(* CoDeSys 2.3.9.41 project: КАРАУЛ 10.07.20.pro *)
(* Libraries: Util.lib 18.5.10 15:14:28, UNM.lib 12.9.19 10:56:53, PID_Regulators.lib 12.9.19 10:56:56, STANDARD.LIB 4.10.05 11:14:46, IECSFC.LIB 13.4.06 15:51:28, SYSLIBTIME.LIB 12.9.19 10:55:25, ANALYZATION.LIB 5.10.99 09:05:06 *)

(* PLC configuration (modules and I/O channels)
SBROS_ALL_ERROR AT %IX0.0 [BitInput] DI_1 {ChannellName = Enter name}
AT %IX0.1 [BitInput] DI_2 {ChannellName = Enter name}
B4_GORELKA_1 AT %IX0.2 [BitInput] DI_3 {ChannellName = Enter name}
B4_GORELKA_2 AT %IX0.3 [BitInput] DI_4 {ChannellName = Enter name}
AT %IB1.0 [ByteInput] 8 discrete inputs {ChannellName = Enter name}
AT %IB1.1 [ByteInput] 4 discrete inputs {ChannellName = Enter name}
ESBE_1_LESS AT %QX2.0 [BitOutput] DO_1 {ChannellName = Enter name}
ESBE_1_MORE AT %QX2.1 [BitOutput] DO_2 {ChannellName = Enter name}
ESBE_2_LESS AT %QX2.2 [BitOutput] DO_3 {ChannellName = Enter name}
ESBE_2_MORE AT %QX2.3 [BitOutput] DO_4 {ChannellName = Enter name}
AT %QB3.0 [ByteOutput] 8 discrete outputs {ChannellName = Enter name}
AT %QB3.1 [ByteOutput] 8 signal outputs {ChannellName = Enter name}
Fast analog inputs [ID125] node 4, in %IB4 out %QB4 {ChannellName = Fast analog inputs; Flt_Comm = 50Hz 2Por}
  AT %IR4.0 [FloatInputP] AI #1 {ChannellName = Fast analog input; AIN_TYPE = 4-20 mA; Peak_Filtr = 200; Flt_Ch = Off; TauRC = 10; MinFV = 0; MaxFV = 20000.0}
  AT %IR4.1 [FloatInputP] AI #2 {ChannellName = Fast analog input; AIN_TYPE = 4-20 mA; Peak_Filtr = 200; Flt_Ch = Off; TauRC = 10; MinFV = 0; MaxFV = 20000.0}
  AT %IR4.2 [FloatInputP] AI #3 {ChannellName = Fast analog input; AIN_TYPE = 4-20 mA; Peak_Filtr = 200; Flt_Ch = Off; TauRC = 10; MinFV = 0; MaxFV = 20000.0}
  AT %IR4.3 [FloatInputP] AI #4 {ChannellName = Fast analog input; AIN_TYPE = 4-20 mA; Peak_Filtr = 200; Flt_Ch = Off; TauRC = 10; MinFV = 0; MaxFV = 20000.0}
  AT %IR4.4 [FloatInputP] AI #5 {ChannellName = Fast analog input; AIN_TYPE = 4-20 mA; Peak_Filtr = 200; Flt_Ch = Off; TauRC = 10; MinFV = 0; MaxFV = 20000.0}
  AT %IR4.5 [FloatInputP] AI #6 {ChannellName = Fast analog input; AIN_TYPE = 4-20 mA; Peak_Filtr = 200; Flt_Ch = Off; TauRC = 10; MinFV = 0; MaxFV = 20000.0}
  AT %IR4.6 [FloatInputP] AI #7 {ChannellName = Fast analog input; AIN_TYPE = 4-20 mA; Peak_Filtr = 200; Flt_Ch = Off; TauRC = 10; MinFV = 0; MaxFV = 20000.0}
  AT %IR4.7 [FloatInputP] AI #8 {ChannellName = Fast analog input; AIN_TYPE = 4-20 mA; Peak_Filtr = 200; Flt_Ch = Off; TauRC = 10; MinFV = 0; MaxFV = 20000.0}
  AT %IW4.8 [WordInput] AI read time (10ms) {ChannellName = Enter name}
Analog outputs [ID126] node 5, in %IB5 out %QB5 {ChannellName = Analog outputs}
  AT %QR5.0 [FloatOutputP] AO #1 {ChannellName = Analog output; AOUT_TYPE = 4-20 mA; SafeValueREAL = 0.0}
  AT %QR5.1 [FloatOutputP] AO #2 {ChannellName = Analog output; AOUT_TYPE = 4-20 mA; SafeValueREAL = 0.0}
  AT %QR5.2 [FloatOutputP] AO #3 {ChannellName = Analog output; AOUT_TYPE = 4-20 mA; SafeValueREAL = 0.0}
  AT %QR5.3 [FloatOutputP] AO #4 {ChannellName = Analog output; AOUT_TYPE = 4-20 mA; SafeValueREAL = 0.0}
Special input [ID103] node 6, in %IB6 out %QB6 {ChannellName = Special input}
  AT %IX6.0 [BitInput] Special input {ChannellName = Enter name}
Special output [ID104] node 7, in %IB7 out %QB7 {ChannellName = Special output}
  AT %QX7.0 [BitOutput] Special output {ChannellName = Enter name}
RS-232 [COM2_USART] node 0, in %IB8.0.0 out %QB8.0.0 {ChannellName = RS-232; CommunicationSpeed = 115200; Parity = NO PARITY CHECK; BitLength = 8 bits; StopLength = One stop bit; InterfaceType = RS232; FrameOriented = RTU; Timeout = 0; Visibility = No}
AT %QB8.1.0 [ByteOutput] {ChannellName = Enter name}
AT %QB8.2.0 [ByteOutput] {ChannellName = Enter name}
AT %QB8.3.0 [ByteOutput] {ChannellName = Enter name}
AT %QB8.4.0 [ByteOutput] {ChannellName = Enter name}
AT %QB8.5.0 [ByteOutput] {ChannellName = Enter name}
AT %QB8.6.0 [ByteOutput] {ChannellName = Enter name}
AT %QB8.7.0 [ByteOutput] {ChannellName = Enter name}
AT %QB8.8.0 [ByteOutput] {ChannellName = Enter name}
AT %QB8.9.0 [ByteOutput] {ChannellName = Enter name}
AT %QB8.10.0 [ByteOutput] {ChannellName = Enter name}
AT %QB8.11.0 [ByteOutput] {ChannellName = Enter name}
AT %QB8.12.0 [ByteOutput] {ChannellName = Enter name}
AT %QB8.13.0 [ByteOutput] {ChannellName = Enter name}
AT %QB8.14.0 [ByteOutput] {ChannellName = Enter name}
AT %QB8.15.0 [ByteOutput] {ChannellName = Enter name}
AT %QB8.16.0 [ByteOutput] {ChannellName = Enter name}
AT %QB8.17.0 [ByteOutput] {ChannellName = Enter name}
AT %QB8.18.0 [ByteOutput] {ChannellName = Enter name}
8 bits [8Bit] node 19, in %IB8.19 out %QB8.19 {ChannellName = 8 bit}
  AT %QB8.19.0 [ByteOutput] {ChannellName = Enter name}
8 bits [8Bit] node 20, in %IB8.20 out %QB8.20 {ChannellName = 8 bit}
  AT %QB8.20.0 [ByteOutput] {ChannellName = Enter name}
AVAR_DAVL_PR_OTOP_MAX AT %QD8.21.0 [FloatOutput] {ChannellName = Enter name}
AVAR_DAVL_PR_OTOP_MIN AT %QD8.22.0 [FloatOutput] {ChannellName = Enter name}
USTAVKA_DAVL_OBR_OTOP_ZIMNIY AT %QD8.23.0 [FloatOutput] {ChannellName = Enter name}
PEREPAD_DAVL_OTOP AT %QD8.24.0 [FloatOutput] {ChannellName = Enter name}
AVAR_VREMA_NASOS_OTOPL AT %QD8.25.0 [FloatOutput] {ChannellName = Enter name}
OSNOVNOY_SETEVOY_NASOS AT %QD8.26.0 [FloatOutput] {ChannellName = Enter name}
GISTEREZIS_PODPITKI_OTOPL AT %QD8.27.0 [FloatOutput] {ChannellName = Enter name}
DAVL_POKOYA_OTOP AT %QD8.28.0 [FloatOutput] {ChannellName = Enter name}
Float [Float] node 29, in %IB8.29 out %QB8.29 {ChannellName = float}
  AT %QD8.29.0 [FloatOutput] {ChannellName = Enter name}
Float [Float] node 30, in %IB8.30 out %QB8.30 {ChannellName = float}
  AT %QD8.30.0 [FloatOutput] {ChannellName = Enter name}
Float [Float] node 31, in %IB8.31 out %QB8.31 {ChannellName = float}
  AT %QD8.31.0 [FloatOutput] {ChannellName = Enter name}
Float [Float] node 32, in %IB8.32 out %QB8.32 {ChannellName = float}
  AT %QD8.32.0 [FloatOutput] {ChannellName = Enter name}
  AVAR_DAVL_PR_GVS_MAX AT %QD8.33.0 [FloatOutput] {ChannellName = Enter name}
  AVAR_DAVL_PR_GVS_MIN AT %QD8.34.0 [FloatOutput] {ChannellName = Enter name}
  USTAVKA_DAVL_OBR_GVS AT %QD8.35.0 [FloatOutput] {ChannellName = Enter name}
  PEREPAD_DAVL_GVS AT %QD8.36.0 [FloatOutput] {ChannellName = Enter name}
  AVAR_VREMA_NASOS_GVS AT %QD8.37.0 [FloatOutput] {ChannellName = Enter name}
  OSNOVNOY_GVS_NASOS AT %QD8.38.0 [FloatOutput] {ChannellName = Enter name}
  GISTEREZIS_PODPITKI_GVS AT %QD8.39.0 [FloatOutput] {ChannellName = Enter name}
  DAVL_POKOYA_GVS AT %QD8.40.0 [FloatOutput] {ChannellName = Enter name}
Float [Float] node 41, in %IB8.41 out %QB8.41 {ChannellName = float}
  AT %QD8.41.0 [FloatOutput] {ChannellName = Enter name}
Float [Float] node 42, in %IB8.42 out %QB8.42 {ChannellName = float}
  AT %QD8.42.0 [FloatOutput] {ChannellName = Enter name}
Float [Float] node 43, in %IB8.43 out %QB8.43 {ChannellName = float}
  AT %QD8.43.0 [FloatOutput] {ChannellName = Enter name}
Float [Float] node 44, in %IB8.44 out %QB8.44 {ChannellName = float}
  AT %QD8.44.0 [FloatOutput] {ChannellName = Enter name}
  Float3Module.MODBUS_ID400Parameter.Chan AT %QD8.45.0 [FloatOutput] ellName1Module.FloatfloatfloatSTRINGFloat-IB-%QB-%MB-%M {ChannellName = Enter name}
  Float3Module.MODBUS_ID400Parameter.Chan AT %QD8.46.0 [FloatOutput] ellName1Module.FloatfloatfloatSTRINGFloat.IB.%QB.%MB.%M {ChannellName = Enter name}
Float [Float] node 47, in %IB8.47 out %QB8.47 {ChannellName = float}
  AT %QD8.47.0 [FloatOutput] {ChannellName = Enter name}
Float [Float] node 48, in %IB8.48 out %QB8.48 {ChannellName = float}
  AT %QD8.48.0 [FloatOutput] {ChannellName = Enter name}
  AVAR_VREMA_NASOS_PODPITKI AT %QD8.49.0 [FloatOutput] {ChannellName = Enter name}
  OSNOVNOY_PODPITOCHNIY_NASOS AT %QD8.50.0 [FloatOutput] {ChannellName = Enter name}
Float [Float] node 51, in %IB8.51 out %QB8.51 {ChannellName = float}
  AT %QD8.51.0 [FloatOutput] {ChannellName = Enter name}
Float [Float] node 52, in %IB8.52 out %QB8.52 {ChannellName = float}
  AT %QD8.52.0 [FloatOutput] {ChannellName = Enter name}
Float [Float] node 53, in %IB8.53 out %QB8.53 {ChannellName = float}
  AT %QD8.53.0 [FloatOutput] {ChannellName = Enter name}
Float [Float] node 54, in %IB8.54 out %QB8.54 {ChannellName = float}
  AT %QD8.54.0 [FloatOutput] {ChannellName = Enter name}
Float [Float] node 55, in %IB8.55 out %QB8.55 {ChannellName = float}
  AT %QD8.55.0 [FloatOutput] {ChannellName = Enter name}
Float [Float] node 56, in %IB8.56 out %QB8.56 {ChannellName = float}
  AT %QD8.56.0 [FloatOutput] {ChannellName = Enter name}
  AVAR_DAVL_PR_VNUTR_MAX AT %QD8.57.0 [FloatOutput] {ChannellName = Enter name}
  AVAR_DAVL_PR_VNUTR_MIN AT %QD8.58.0 [FloatOutput] {ChannellName = Enter name}
  USTAVKA_DAVL_OBR_VNUTR AT %QD8.59.0 [FloatOutput] {ChannellName = Enter name}
  PEREPAD_DAVL_VNUTR AT %QD8.60.0 [FloatOutput] {ChannellName = Enter name}
  AVAR_VREMA_NASOS_VNUTR AT %QD8.61.0 [FloatOutput] {ChannellName = Enter name}
  OSNOVNOY_VNUTR_NASOS AT %QD8.62.0 [FloatOutput] {ChannellName = Enter name}
  GISTEREZIS_PODPITKI_VNUTR AT %QD8.63.0 [FloatOutput] {ChannellName = Enter name}
  DAVL_POKOYA_VNUTR AT %QD8.64.0 [FloatOutput] {ChannellName = Enter name}
Float [Float] node 65, in %IB8.65 out %QB8.65 {ChannellName = float}
  AT %QD8.65.0 [FloatOutput] {ChannellName = Enter name}
Float [Float] node 66, in %IB8.66 out %QB8.66 {ChannellName = float}
  AT %QD8.66.0 [FloatOutput] {ChannellName = Enter name}
Float [Float] node 67, in %IB8.67 out %QB8.67 {ChannellName = float}
  AT %QD8.67.0 [FloatOutput] {ChannellName = Enter name}
Float [Float] node 68, in %IB8.68 out %QB8.68 {ChannellName = float}
  AT %QD8.68.0 [FloatOutput] {ChannellName = Enter name}
Float [Float] node 69, in %IB8.69 out %QB8.69 {ChannellName = float}
  VREMYA_RABOTU_CIRCULYACIONNOGO_NASOSA AT %QD8.69.0 [FloatOutput] {ChannellName = Enter name}
Float [Float] node 70, in %IB8.70 out %QB8.70 {ChannellName = float}
  TEMPERATURA_OFF_CIRCULACIONNOGO_NASOSA AT %QD8.70.0 [FloatOutput] {ChannellName = Enter name}
  OSNOVNAYA_GORELKA AT %QD8.71.0 [FloatOutput] {ChannellName = Enter name}
  PODOGREV_2_GORELKOY AT %QD8.72.0 [FloatOutput] {ChannellName = Enter name}
Float [Float] node 73, in %IB8.73 out %QB8.73 {ChannellName = float}
  TEMPERATURA_VKLUCHENIYA_GORELKA_1 AT %QD8.73.0 [FloatOutput] {ChannellName = Enter name}
Float [Float] node 74, in %IB8.74 out %QB8.74 {ChannellName = float}
  TEMPERATURA_OFF_2_STUPENI_GORELKA_1 AT %QD8.74.0 [FloatOutput] {ChannellName = Enter name}
Float [Float] node 75, in %IB8.75 out %QB8.75 {ChannellName = float}
  TEMPERATURA_OFF_TERMOSTAT_GORELKA_1 AT %QD8.75.0 [FloatOutput] {ChannellName = Enter name}
Float [Float] node 76, in %IB8.76 out %QB8.76 {ChannellName = float}
  GISTEREZIS_1_2_STUPEN_GORELKA_1 AT %QD8.76.0 [FloatOutput] {ChannellName = Enter name}
Float [Float] node 77, in %IB8.77 out %QB8.77 {ChannellName = float}
  VREMYA_SBROS_AVARIA_GORELKA_1 AT %QD8.77.0 [FloatOutput] {ChannellName = Enter name}
Float [Float] node 78, in %IB8.78 out %QB8.78 {ChannellName = float}
  TEMPERATURA_AVARIA_MAX_GORELKA_1 AT %QD8.78.0 [FloatOutput] {ChannellName = Enter name}
Float [Float] node 79, in %IB8.79 out %QB8.79 {ChannellName = float}
  AT %QD8.79.0 [FloatOutput] {ChannellName = Enter name}
Float [Float] node 80, in %IB8.80 out %QB8.80 {ChannellName = float}
  AT %QD8.80.0 [FloatOutput] {ChannellName = Enter name}
  PODOGREV_3_GORELKOY AT %QD8.81.0 [FloatOutput] {ChannellName = Enter name}
Float [Float] node 82, in %IB8.82 out %QB8.82 {ChannellName = float}
  TEMPERATURA_VKLUCHENIYA_GORELKA_2 AT %QD8.82.0 [FloatOutput] {ChannellName = Enter name}
Float [Float] node 83, in %IB8.83 out %QB8.83 {ChannellName = float}
  TEMPERATURA_OFF_2_STUPENI_GORELKA_2 AT %QD8.83.0 [FloatOutput] {ChannellName = Enter name}
Float [Float] node 84, in %IB8.84 out %QB8.84 {ChannellName = float}
  TEMPERATURA_OFF_TERMOSTAT_GORELKA_2 AT %QD8.84.0 [FloatOutput] {ChannellName = Enter name}
Float [Float] node 85, in %IB8.85 out %QB8.85 {ChannellName = float}
  GISTEREZIS_1_2_STUPEN_GORELKA_2 AT %QD8.85.0 [FloatOutput] {ChannellName = Enter name}
Float [Float] node 86, in %IB8.86 out %QB8.86 {ChannellName = float}
  VREMYA_SBROS_AVARIA_GORELKA_2 AT %QD8.86.0 [FloatOutput] {ChannellName = Enter name}
  TEMPERATURA_AVARIA_MAX_GORELKA_2 AT %QD8.87.0 [FloatOutput] {ChannellName = Enter name}
Float [Float] node 88, in %IB8.88 out %QB8.88 {ChannellName = float}
  AT %QD8.88.0 [FloatOutput] {ChannellName = Enter name}
Float [Float] node 89, in %IB8.89 out %QB8.89 {ChannellName = float}
  AT %QD8.89.0 [FloatOutput] {ChannellName = Enter name}
Float [Float] node 90, in %IB8.90 out %QB8.90 {ChannellName = float}
  AT %QD8.90.0 [FloatOutput] {ChannellName = Enter name}
Float [Float] node 91, in %IB8.91 out %QB8.91 {ChannellName = float}
  AT %QD8.91.0 [FloatOutput] {ChannellName = Enter name}
Float [Float] node 92, in %IB8.92 out %QB8.92 {ChannellName = float}
  AT %QD8.92.0 [FloatOutput] {ChannellName = Enter name}
Float [Float] node 93, in %IB8.93 out %QB8.93 {ChannellName = float}
  AT %QD8.93.0 [FloatOutput] {ChannellName = Enter name}
Float [Float] node 94, in %IB8.94 out %QB8.94 {ChannellName = float}
  AT %QD8.94.0 [FloatOutput] {ChannellName = Enter name}
Float [Float] node 95, in %IB8.95 out %QB8.95 {ChannellName = float}
  AT %QD8.95.0 [FloatOutput] {ChannellName = Enter name}
Float [Float] node 96, in %IB8.96 out %QB8.96 {ChannellName = float}
  TEMPERATURA_AVARIA_MAX_GORELKA_3 AT %QD8.96.0 [FloatOutput] {ChannellName = Enter name}
Float [Float] node 97, in %IB8.97 out %QB8.97 {ChannellName = float}
  SECOND_GORELKA AT %QD8.97.0 [FloatOutput] {ChannellName = Enter name}
Float [Float] node 98, in %IB8.98 out %QB8.98 {ChannellName = float}
  RESERV_GORELKA AT %QD8.98.0 [FloatOutput] {ChannellName = Enter name}
  GISTEREZIS_PODOGREV AT %QD8.99.0 [FloatOutput] {ChannellName = Enter name}
Float [Float] node 100, in %IB8.100 out %QB8.100 {ChannellName = float}
  AT %QD8.100.0 [FloatOutput] {ChannellName = Enter name}
Float [Float] node 101, in %IB8.101 out %QB8.101 {ChannellName = float}
  AT %QD8.101.0 [FloatOutput] {ChannellName = Enter name}
Float [Float] node 102, in %IB8.102 out %QB8.102 {ChannellName = float}
  AT %QD8.102.0 [FloatOutput] {ChannellName = Enter name}
Float [Float] node 103, in %IB8.103 out %QB8.103 {ChannellName = float}
  AT %QD8.103.0 [FloatOutput] {ChannellName = Enter name}
Float [Float] node 104, in %IB8.104 out %QB8.104 {ChannellName = float}
  AT %QD8.104.0 [FloatOutput] {ChannellName = Enter name}
Float [Float] node 105, in %IB8.105 out %QB8.105 {ChannellName = float}
  AT %QD8.105.0 [FloatOutput] {ChannellName = Enter name}
Float [Float] node 106, in %IB8.106 out %QB8.106 {ChannellName = float}
  AT %QD8.106.0 [FloatOutput] {ChannellName = Enter name}
Float [Float] node 107, in %IB8.107 out %QB8.107 {ChannellName = float}
  AT %QD8.107.0 [FloatOutput] {ChannellName = Enter name}
Float [Float] node 108, in %IB8.108 out %QB8.108 {ChannellName = float}
  AT %QD8.108.0 [FloatOutput] {ChannellName = Enter name}
Float [Float] node 109, in %IB8.109 out %QB8.109 {ChannellName = float}
  AT %QD8.109.0 [FloatOutput] {ChannellName = Enter name}
Float [Float] node 110, in %IB8.110 out %QB8.110 {ChannellName = float}
  AT %QD8.110.0 [FloatOutput] {ChannellName = Enter name}
Float [Float] node 111, in %IB8.111 out %QB8.111 {ChannellName = float}
  AT %QD8.111.0 [FloatOutput] {ChannellName = Enter name}
  EL_2_DAVL_SBROSA_PR_OTOP AT %QD8.112.0 [FloatOutput] {ChannellName = Enter name}
  GISTEREZIS_SBROS_OTOPLENIYA AT %QD8.113.0 [FloatOutput] {ChannellName = Enter name}
Float [Float] node 114, in %IB8.114 out %QB8.114 {ChannellName = float}
  AT %QD8.114.0 [FloatOutput] {ChannellName = Enter name}
  EL_3_DAVL_SBROSA_GVS AT %QD8.115.0 [FloatOutput] {ChannellName = Enter name}
  GISTEREZIS_SBROS_GVS AT %QD8.116.0 [FloatOutput] {ChannellName = Enter name}
Float [Float] node 117, in %IB8.117 out %QB8.117 {ChannellName = float}
  AT %QD8.117.0 [FloatOutput] {ChannellName = Enter name}
Float [Float] node 118, in %IB8.118 out %QB8.118 {ChannellName = float}
  AT %QD8.118.0 [FloatOutput] {ChannellName = Enter name}
Float [Float] node 119, in %IB8.119 out %QB8.119 {ChannellName = float}
  AT %QD8.119.0 [FloatOutput] {ChannellName = Enter name}
Float [Float] node 120, in %IB8.120 out %QB8.120 {ChannellName = float}
  AT %QD8.120.0 [FloatOutput] {ChannellName = Enter name}
Float [Float] node 121, in %IB8.121 out %QB8.121 {ChannellName = float}
  AT %QD8.121.0 [FloatOutput] {ChannellName = Enter name}
Float [Float] node 122, in %IB8.122 out %QB8.122 {ChannellName = float}
  AT %QD8.122.0 [FloatOutput] {ChannellName = Enter name}
Float [Float] node 123, in %IB8.123 out %QB8.123 {ChannellName = float}
  AT %QD8.123.0 [FloatOutput] {ChannellName = Enter name}
Float [Float] node 124, in %IB8.124 out %QB8.124 {ChannellName = float}
  PROPORCIONALNAYA_SOSTAV_ESBE_1 AT %QD8.124.0 [FloatOutput] {ChannellName = Enter name}
Float [Float] node 125, in %IB8.125 out %QB8.125 {ChannellName = float}
  INTEGRALNAYA_SOSTAV_ESBE_1 AT %QD8.125.0 [FloatOutput] {ChannellName = Enter name}
Float [Float] node 126, in %IB8.126 out %QB8.126 {ChannellName = float}
  DIFFERENCIALNAYA_SOSTAV_ESBE_1 AT %QD8.126.0 [FloatOutput] {ChannellName = Enter name}
Float [Float] node 127, in %IB8.127 out %QB8.127 {ChannellName = float}
  VREMYA_HODA_ZADVIZKI_ESBE_1 AT %QD8.127.0 [FloatOutput] {ChannellName = Enter name}
Float [Float] node 128, in %IB8.128 out %QB8.128 {ChannellName = float}
  MIN_VREMYA_OSTANOVKI_ESBE_1 AT %QD8.128.0 [FloatOutput] {ChannellName = Enter name}
Float [Float] node 129, in %IB8.129 out %QB8.129 {ChannellName = float}
  MIN_VREMYA_HODA_ESBE_1 AT %QD8.129.0 [FloatOutput] {ChannellName = Enter name}
  KORREKTIROVKA_USTAVKI_ESBE_1 AT %QD8.130.0 [FloatOutput] {ChannellName = Enter name}
  PROCENT_OTKLONENIA_OT_USTAVKI_ESBE_1 AT %QD8.131.0 [FloatOutput] {ChannellName = Enter name}
  VREMYA_OZIDANIYA_POSLE_SBROSA_ESBE_1 AT %QD8.132.0 [FloatOutput] {ChannellName = Enter name}
  USTAVKA_POSTOYANNAYA_ESBE_1 AT %QD8.133.0 [FloatOutput] {ChannellName = Enter name}
  PROPORCIONALNAYA_SOSTAV_ESBE_2 AT %QD8.134.0 [FloatOutput] {ChannellName = Enter name}
  INTEGRALNAYA_SOSTAV_ESBE_2 AT %QD8.135.0 [FloatOutput] {ChannellName = Enter name}
  DIFFERENCIALNAYA_SOSTAV_ESBE_2 AT %QD8.136.0 [FloatOutput] {ChannellName = Enter name}
  VREMYA_HODA_ZADVIZKI_ESBE_2 AT %QD8.137.0 [FloatOutput] {ChannellName = Enter name}
  MIN_VREMYA_OSTANOVKI_ESBE_2 AT %QD8.138.0 [FloatOutput] {ChannellName = Enter name}
  MIN_VREMYA_HODA_ESBE_2 AT %QD8.139.0 [FloatOutput] {ChannellName = Enter name}
  KORREKTIROVKA_USTAVKI_ESBE_2 AT %QD8.140.0 [FloatOutput] {ChannellName = Enter name}
  PROCENT_OTKLONENIA_OT_USTAVKI_ESBE_2 AT %QD8.141.0 [FloatOutput] {ChannellName = Enter name}
  VREMYA_OZIDANIYA_POSLE_SBROSA_ESBE_2 AT %QD8.142.0 [FloatOutput] {ChannellName = Enter name}
  USTAVKA_POSTOYANNAYA_ESBE_2 AT %QD8.143.0 [FloatOutput] {ChannellName = Enter name}
  BAK_NIGNAYA_GRANICA AT %QD8.144.0 [FloatOutput] {ChannellName = Enter name}
  BAK_VERHNYAY_GRANICA AT %QD8.145.0 [FloatOutput] {ChannellName = Enter name}
  BAK_MIN_PROCENT_AVARIA AT %QD8.146.0 [FloatOutput] {ChannellName = Enter name}
  BAK_MAX_PROCENT_AVARIA AT %QD8.147.0 [FloatOutput] {ChannellName = Enter name}
  BAK_USTAVKA_NAPOLNENIA AT %QD8.148.0 [FloatOutput] {ChannellName = Enter name}
  BAK_GISTEREZIS_NAPOLNENIA AT %QD8.149.0 [FloatOutput] {ChannellName = Enter name}
Float [Float] node 150, in %IB8.150 out %QB8.150 {ChannellName = float}
  AT %QD8.150.0 [FloatOutput] {ChannellName = Enter name}
Float [Float] node 151, in %IB8.151 out %QB8.151 {ChannellName = float}
  AT %QD8.151.0 [FloatOutput] {ChannellName = Enter name}
  NARABOTKA_MINUT_KASKAD_1_NASOS_1_SETEVOY_SP_307 AT %QD8.152.0 [FloatOutput] {ChannellName = Enter name}
  NARABOTKA_MINUT_KASKAD_1_NASOS_2_SETEVOY_SP_307 AT %QD8.153.0 [FloatOutput] {ChannellName = Enter name}
  NARABOTKA_MINUT_KASKAD_3_NASOS_1_GVS_SP_307 AT %QD8.154.0 [FloatOutput] {ChannellName = Enter name}
  NARABOTKA_MINUT_KASKAD_3_NASOS_2_GVS_SP_307 AT %QD8.155.0 [FloatOutput] {ChannellName = Enter name}
  NARABOTKA_MINUT_KASKAD_4_NASOS_1_PODPITKA_SP_307 AT %QD8.156.0 [FloatOutput] {ChannellName = Enter name}
  NARABOTKA_MINUT_KASKAD_4_NASOS_2_PODPITKA_SP_307 AT %QD8.157.0 [FloatOutput] {ChannellName = Enter name}
  NARABOTKA_MINUT_KASKAD_5_NASOS_1_CIRKUL_SP_307 AT %QD8.158.0 [FloatOutput] {ChannellName = Enter name}
  NARABOTKA_MINUT_KASKAD_5_NASOS_2_CIRKUL_SP_307 AT %QD8.159.0 [FloatOutput] {ChannellName = Enter name}
  NARABOTKA_MINUT_GORELKA_1_SP_307 AT %QD8.160.0 [FloatOutput] {ChannellName = Enter name}
Float [Float] node 161, in %IB8.161 out %QB8.161 {ChannellName = float}
  NARABOTKA_MINUT_GORELKA_2_SP_307 AT %QD8.161.0 [FloatOutput] {ChannellName = Enter name}
Float [Float] node 162, in %IB8.162 out %QB8.162 {ChannellName = float}
  NARABOTKA_MINUT_KASKAD_2_VNUTR_NASOS_1_SP_307 AT %QD8.162.0 [FloatOutput] {ChannellName = Enter name}
Float [Float] node 163, in %IB8.163 out %QB8.163 {ChannellName = float}
  NARABOTKA_MINUT_KASKAD_2_VNUTR_NASOS_2_SP_307 AT %QD8.163.0 [FloatOutput] {ChannellName = Enter name}
Float [Float] node 164, in %IB8.164 out %QB8.164 {ChannellName = float}
  NARABOTKA_MINUT_KASKAD_5_NASOS_3_CIRKUL_SP_307 AT %QD8.164.0 [FloatOutput] {ChannellName = Enter name}
Float [Float] node 165, in %IB8.165 out %QB8.165 {ChannellName = float}
  NARABOTKA_MINUT_GORELKA_3_SP_307 AT %QD8.165.0 [FloatOutput] {ChannellName = Enter name}
Float [Float] node 166, in %IB8.166 out %QB8.166 {ChannellName = float}
  KOLICHESTVO_VKLUCHENIY_KASKAD_1_NASOS_1_SETEVOY_SP_307 AT %QD8.166.0 [FloatOutput] {ChannellName = Enter name}
Float [Float] node 167, in %IB8.167 out %QB8.167 {ChannellName = float}
  KOLICHESTVO_VKLUCHENIY_KASKAD_1_NASOS_2_SETEVOY_SP_307 AT %QD8.167.0 [FloatOutput] {ChannellName = Enter name}
Float [Float] node 168, in %IB8.168 out %QB8.168 {ChannellName = float}
  KOLICHESTVO_VKLUCHENIY_KASKAD_3_NASOS_1_GVS_SP_307 AT %QD8.168.0 [FloatOutput] {ChannellName = Enter name}
Float [Float] node 169, in %IB8.169 out %QB8.169 {ChannellName = float}
  KOLICHESTVO_VKLUCHENIY_KASKAD_3_NASOS_2_GVS_SP_307 AT %QD8.169.0 [FloatOutput] {ChannellName = Enter name}
Float [Float] node 170, in %IB8.170 out %QB8.170 {ChannellName = float}
  KOLICHESTVO_VKLUCHENIY_KASKAD_4_NASOS_1_PODPITKA_SP_307 AT %QD8.170.0 [FloatOutput] {ChannellName = Enter name}
Float [Float] node 171, in %IB8.171 out %QB8.171 {ChannellName = float}
  KOLICHESTVO_VKLUCHENIY_KASKAD_4_NASOS_2_PODPITKA_SP_307 AT %QD8.171.0 [FloatOutput] {ChannellName = Enter name}
Float [Float] node 172, in %IB8.172 out %QB8.172 {ChannellName = float}
  KOLICHESTVO_VKLUCHENIY_KASKAD_5_NASOS_1_CIRKUL_SP_307 AT %QD8.172.0 [FloatOutput] {ChannellName = Enter name}
Float [Float] node 173, in %IB8.173 out %QB8.173 {ChannellName = float}
  KOLICHESTVO_VKLUCHENIY_KASKAD_5_NASOS_2_CIRKUL_SP_307 AT %QD8.173.0 [FloatOutput] {ChannellName = Enter name}
Float [Float] node 174, in %IB8.174 out %QB8.174 {ChannellName = float}
  KOLICHESTVO_VKLUCHENIY_GORELKA_1_SP_307 AT %QD8.174.0 [FloatOutput] {ChannellName = Enter name}
Float [Float] node 175, in %IB8.175 out %QB8.175 {ChannellName = float}
  KOLICHESTVO_VKLUCHENIY_GORELKA_2_SP_307 AT %QD8.175.0 [FloatOutput] {ChannellName = Enter name}
Float [Float] node 176, in %IB8.176 out %QB8.176 {ChannellName = float}
  KOLICHESTVO_VKLUCHENIY_KASKAD_2_VNUTR_NASOS_1_SP_307 AT %QD8.176.0 [FloatOutput] {ChannellName = Enter name}
Float [Float] node 177, in %IB8.177 out %QB8.177 {ChannellName = float}
  KOLICHESTVO_VKLUCHENIY_KASKAD_2_VNUTR_NASOS_2_SP_307 AT %QD8.177.0 [FloatOutput] {ChannellName = Enter name}
Float [Float] node 178, in %IB8.178 out %QB8.178 {ChannellName = float}
  KOLICHESTVO_VKLUCHENIY_KASKAD_5_NASOS_3_CIRKUL_SP_307 AT %QD8.178.0 [FloatOutput] {ChannellName = Enter name}
Float [Float] node 179, in %IB8.179 out %QB8.179 {ChannellName = float}
  KOLICHESTVO_VKLUCHENIY_GORELKA_3_SP_307 AT %QD8.179.0 [FloatOutput] {ChannellName = Enter name}
Float [Float] node 180, in %IB8.180 out %QB8.180 {ChannellName = float}
  TEL_KOD_1 AT %QD8.180.0 [FloatOutput] {ChannellName = Enter name}
  TEL_NOMER_1 AT %QD8.181.0 [FloatOutput] {ChannellName = Enter name}
  TEL_KOD_2 AT %QD8.182.0 [FloatOutput] {ChannellName = Enter name}
  TEL_NOMER_2 AT %QD8.183.0 [FloatOutput] {ChannellName = Enter name}
  TEL_KOD_3 AT %QD8.184.0 [FloatOutput] {ChannellName = Enter name}
  TEL_NOMER_3 AT %QD8.185.0 [FloatOutput] {ChannellName = Enter name}
  KOLICESTVO_SOOBSHENIY AT %QD8.186.0 [FloatOutput] {ChannellName = Enter name}
  KOLICHESTVO_NOMEROV AT %QD8.187.0 [FloatOutput] {ChannellName = Enter name}
  TIME_PLANOVAYA_REBBOT_MODEM AT %QD8.188.0 [FloatOutput] {ChannellName = Enter name}
  TIME_WATCH_DOG AT %QD8.189.0 [FloatOutput] {ChannellName = Enter name}
Float [Float] node 190, in %IB8.190 out %QB8.190 {ChannellName = float}
  AT %QD8.190.0 [FloatOutput] {ChannellName = Enter name}
Float [Float] node 191, in %IB8.191 out %QB8.191 {ChannellName = float}
  AT %QD8.191.0 [FloatOutput] {ChannellName = Enter name}
  VREMYA_ZADERGKI_OBRUV_DATCHIKA AT %QD8.192.0 [FloatOutput] {ChannellName = Enter name}
  VREMYA_ZADERGKI_AVARIA_NIZKOE_DAVLENIE AT %QD8.193.0 [FloatOutput] {ChannellName = Enter name}
Float [Float] node 194, in %IB8.194 out %QB8.194 {ChannellName = float}
  AT %QD8.194.0 [FloatOutput] {ChannellName = Enter name}
Float [Float] node 195, in %IB8.195 out %QB8.195 {ChannellName = float}
  AT %QD8.195.0 [FloatOutput] {ChannellName = Enter name}
Float [Float] node 196, in %IB8.196 out %QB8.196 {ChannellName = float}
  AT %QD8.196.0 [FloatOutput] {ChannellName = Enter name}
Float [Float] node 197, in %IB8.197 out %QB8.197 {ChannellName = float}
  AT %QD8.197.0 [FloatOutput] {ChannellName = Enter name}
Float [Float] node 198, in %IB8.198 out %QB8.198 {ChannellName = float}
  TEMPERATURA_1_PR_OTOPLENIYA_AI_SP_307 AT %QD8.198.0 [FloatOutput] {ChannellName = Enter name}
Float [Float] node 199, in %IB8.199 out %QB8.199 {ChannellName = float}
  TEMPERATURA_2_OBR_OTOPLENIYA_AI_SP_307 AT %QD8.199.0 [FloatOutput] {ChannellName = Enter name}
Float [Float] node 200, in %IB8.200 out %QB8.200 {ChannellName = float}
  TEMPERATURA_3_PR_GVS_AI_SP_307 AT %QD8.200.0 [FloatOutput] {ChannellName = Enter name}
Float [Float] node 201, in %IB8.201 out %QB8.201 {ChannellName = float}
  TEMPERATURA_4_OBR_GVS_AI_SP_307 AT %QD8.201.0 [FloatOutput] {ChannellName = Enter name}
Float [Float] node 202, in %IB8.202 out %QB8.202 {ChannellName = float}
  TEMPERATURA_5_KOTEL_1_AI_SP_307 AT %QD8.202.0 [FloatOutput] {ChannellName = Enter name}
Float [Float] node 203, in %IB8.203 out %QB8.203 {ChannellName = float}
  TEMPERATURA_6_KOTEL_2_AI_SP_307 AT %QD8.203.0 [FloatOutput] {ChannellName = Enter name}
Float [Float] node 204, in %IB8.204 out %QB8.204 {ChannellName = float}
  TEMPERATURA_7_KOTEL_3_AI_SP_307 AT %QD8.204.0 [FloatOutput] {ChannellName = Enter name}
Float [Float] node 205, in %IB8.205 out %QB8.205 {ChannellName = float}
  TEMPERATURA_8_ULICA_AI_SP_307 AT %QD8.205.0 [FloatOutput] {ChannellName = Enter name}
Float [Float] node 206, in %IB8.206 out %QB8.206 {ChannellName = float}
  DAVLENIE_1_PR_OTOPLENIYA_AI_SP_307 AT %QD8.206.0 [FloatOutput] {ChannellName = Enter name}
Float [Float] node 207, in %IB8.207 out %QB8.207 {ChannellName = float}
  DAVLENIE_2_OBR_OTOPLENIYA_AI_SP_307 AT %QD8.207.0 [FloatOutput] {ChannellName = Enter name}
Float [Float] node 208, in %IB8.208 out %QB8.208 {ChannellName = float}
  DAVLENIE_3_PR_GVS_AI_SP_307 AT %QD8.208.0 [FloatOutput] {ChannellName = Enter name}
Float [Float] node 209, in %IB8.209 out %QB8.209 {ChannellName = float}
  DAVLENIE_4_OBR_GVS_AI_SP_307 AT %QD8.209.0 [FloatOutput] {ChannellName = Enter name}
Float [Float] node 210, in %IB8.210 out %QB8.210 {ChannellName = float}
  DAVLENIE_5_PR_VNUTR_AI_SP_307 AT %QD8.210.0 [FloatOutput] {ChannellName = Enter name}
Float [Float] node 211, in %IB8.211 out %QB8.211 {ChannellName = float}
  DAVLENIE_6_OBR_VNUTR_AI_SP_307 AT %QD8.211.0 [FloatOutput] {ChannellName = Enter name}
Float [Float] node 212, in %IB8.212 out %QB8.212 {ChannellName = float}
  DAVLENIE_7_NAKOPITELNIY_BAK_AI_SP_307 AT %QD8.212.0 [FloatOutput] {ChannellName = Enter name}
Float [Float] node 213, in %IB8.213 out %QB8.213 {ChannellName = float}
  AT %QD8.213.0 [FloatOutput] {ChannellName = Enter name}
Float [Float] node 214, in %IB8.214 out %QB8.214 {ChannellName = float}
  USTAVKA_ESBE_1_SP_307 AT %QD8.214.0 [FloatOutput] {ChannellName = Enter name}
Float [Float] node 215, in %IB8.215 out %QB8.215 {ChannellName = float}
  USTAVKA_ESBE_2_SP_307 AT %QD8.215.0 [FloatOutput] {ChannellName = Enter name}
Float [Float] node 216, in %IB8.216 out %QB8.216 {ChannellName = float}
  AT %QD8.216.0 [FloatOutput] {ChannellName = Enter name}
Float [Float] node 217, in %IB8.217 out %QB8.217 {ChannellName = float}
  AT %QD8.217.0 [FloatOutput] {ChannellName = Enter name}
Float [Float] node 218, in %IB8.218 out %QB8.218 {ChannellName = float}
  AT %QD8.218.0 [FloatOutput] {ChannellName = Enter name}
Float [Float] node 219, in %IB8.219 out %QB8.219 {ChannellName = float}
  AT %QD8.219.0 [FloatOutput] {ChannellName = Enter name}
2 byte [Register] node 220, in %IB8.220 out %QB8.220 {ChannellName = 2 byte}
  STATUS_NASOS_1_SETEVOY_1_SP_307 AT %QW8.220.0 [WordOutput] {ChannellName = Enter name}
2 byte [Register] node 221, in %IB8.221 out %QB8.221 {ChannellName = 2 byte}
  STATUS_NASOS_2_SETEVOY_1_SP_307 AT %QW8.221.0 [WordOutput] {ChannellName = Enter name}
2 byte [Register] node 222, in %IB8.222 out %QB8.222 {ChannellName = 2 byte}
  STATUS_NASOS_LETNIY_SETEVOY_2_SP_307 AT %QW8.222.0 [WordOutput] {ChannellName = Enter name}
2 byte [Register] node 223, in %IB8.223 out %QB8.223 {ChannellName = 2 byte}
  STATUS_TRUBA_SETEVAYA_SP_307 AT %QW8.223.0 [WordOutput] {ChannellName = Enter name}
2 byte [Register] node 224, in %IB8.224 out %QB8.224 {ChannellName = 2 byte}
  STATUS_NASOS_1_GVS_3_SP_307 AT %QW8.224.0 [WordOutput] {ChannellName = Enter name}
2 byte [Register] node 225, in %IB8.225 out %QB8.225 {ChannellName = 2 byte}
  STATUS_NASOS_2_GVS_3_SP_307 AT %QW8.225.0 [WordOutput] {ChannellName = Enter name}
2 byte [Register] node 226, in %IB8.226 out %QB8.226 {ChannellName = 2 byte}
  STATUS_TRUBA_GVS_SP_307 AT %QW8.226.0 [WordOutput] {ChannellName = Enter name}
2 byte [Register] node 227, in %IB8.227 out %QB8.227 {ChannellName = 2 byte}
  STATUS_NASOS_1_PODPIT_4_SP_307 AT %QW8.227.0 [WordOutput] {ChannellName = Enter name}
2 byte [Register] node 228, in %IB8.228 out %QB8.228 {ChannellName = 2 byte}
  STATUS_NASOS_2_PODPIT_4_SP_307 AT %QW8.228.0 [WordOutput] {ChannellName = Enter name}
2 byte [Register] node 229, in %IB8.229 out %QB8.229 {ChannellName = 2 byte}
  STATUS_TRUBA_PODPITKA_SP_307 AT %QW8.229.0 [WordOutput] {ChannellName = Enter name}
2 byte [Register] node 230, in %IB8.230 out %QB8.230 {ChannellName = 2 byte}
  STATUS_NASOS_1_CIRCULAYCIONNUY_SP_307 AT %QW8.230.0 [WordOutput] {ChannellName = Enter name}
2 byte [Register] node 231, in %IB8.231 out %QB8.231 {ChannellName = 2 byte}
  STATUS_NASOS_2_CIRCULAYCIONNUY_SP_307 AT %QW8.231.0 [WordOutput] {ChannellName = Enter name}
2 byte [Register] node 232, in %IB8.232 out %QB8.232 {ChannellName = 2 byte}
  STATUS_NASOS_3_CIRCULAYCIONNUY_SP_307 AT %QW8.232.0 [WordOutput] {ChannellName = Enter name}
2 byte [Register] node 233, in %IB8.233 out %QB8.233 {ChannellName = 2 byte}
  AT %QW8.233.0 [WordOutput] {ChannellName = Enter name}
2 byte [Register] node 234, in %IB8.234 out %QB8.234 {ChannellName = 2 byte}
  AT %QW8.234.0 [WordOutput] {ChannellName = Enter name}
2 byte [Register] node 235, in %IB8.235 out %QB8.235 {ChannellName = 2 byte}
  AT %QW8.235.0 [WordOutput] {ChannellName = Enter name}
2 byte [Register] node 236, in %IB8.236 out %QB8.236 {ChannellName = 2 byte}
  STATUS_GORELKA1_SP_307 AT %QW8.236.0 [WordOutput] {ChannellName = Enter name}
2 byte [Register] node 237, in %IB8.237 out %QB8.237 {ChannellName = 2 byte}
  STATUS_GORELKA2_SP_307 AT %QW8.237.0 [WordOutput] {ChannellName = Enter name}
2 byte [Register] node 238, in %IB8.238 out %QB8.238 {ChannellName = 2 byte}
  STATUS_GORELKA3_SP_307 AT %QW8.238.0 [WordOutput] {ChannellName = Enter name}
2 byte [Register] node 239, in %IB8.239 out %QB8.239 {ChannellName = 2 byte}
  STATUS_GORENIE_1_B_M_SP_307 AT %QW8.239.0 [WordOutput] {ChannellName = Enter name}
2 byte [Register] node 240, in %IB8.240 out %QB8.240 {ChannellName = 2 byte}
  STATUS_GORENIE_2_B_M_SP_307 AT %QW8.240.0 [WordOutput] {ChannellName = Enter name}
2 byte [Register] node 241, in %IB8.241 out %QB8.241 {ChannellName = 2 byte}
  STATUS_GORENIE_3_B_M_SP_307 AT %QW8.241.0 [WordOutput] {ChannellName = Enter name}
2 byte [Register] node 242, in %IB8.242 out %QB8.242 {ChannellName = 2 byte}
  AT %QW8.242.0 [WordOutput] {ChannellName = Enter name}
2 byte [Register] node 243, in %IB8.243 out %QB8.243 {ChannellName = 2 byte}
  AT %QW8.243.0 [WordOutput] {ChannellName = Enter name}
2 byte [Register] node 244, in %IB8.244 out %QB8.244 {ChannellName = 2 byte}
  AT %QW8.244.0 [WordOutput] {ChannellName = Enter name}
2 byte [Register] node 245, in %IB8.245 out %QB8.245 {ChannellName = 2 byte}
  STATUS_EL_KL_1_PODPITKA_SP_307 AT %QW8.245.0 [WordOutput] {ChannellName = Enter name}
2 byte [Register] node 246, in %IB8.246 out %QB8.246 {ChannellName = 2 byte}
  STATUS_EL_KL_2_SBROS_OTOPLENIAYA_SP_307 AT %QW8.246.0 [WordOutput] {ChannellName = Enter name}
2 byte [Register] node 247, in %IB8.247 out %QB8.247 {ChannellName = 2 byte}
  STATUS_EL_KL_3_SBROS_GVS_SP_307 AT %QW8.247.0 [WordOutput] {ChannellName = Enter name}
  STATUS_EL_KL_4_NAK_BAK_SP_307 AT %QW8.248.0 [WordOutput] {ChannellName = Enter name}
2 byte [Register] node 249, in %IB8.249 out %QB8.249 {ChannellName = 2 byte}
  AT %QW8.249.0 [WordOutput] {ChannellName = Enter name}
2 byte [Register] node 250, in %IB8.250 out %QB8.250 {ChannellName = 2 byte}
  AT %QW8.250.0 [WordOutput] {ChannellName = Enter name}
2 byte [Register] node 251, in %IB8.251 out %QB8.251 {ChannellName = 2 byte}
  AT %QW8.251.0 [WordOutput] {ChannellName = Enter name}
2 byte [Register] node 252, in %IB8.252 out %QB8.252 {ChannellName = 2 byte}
  AT %QW8.252.0 [WordOutput] {ChannellName = Enter name}
2 byte [Register] node 253, in %IB8.253 out %QB8.253 {ChannellName = 2 byte}
  STATUS_BAK_PROCENT_ZAPOLNENIA AT %QW8.253.0 [WordOutput] {ChannellName = Enter name}
2 byte [Register] node 254, in %IB8.254 out %QB8.254 {ChannellName = 2 byte}
  STATUS_ESBE_1_SP_307 AT %QW8.254.0 [WordOutput] {ChannellName = Enter name}
2 byte [Register] node 255, in %IB8.255 out %QB8.255 {ChannellName = 2 byte}
  STATUS_ESBE_2_SP_307 AT %QW8.255.0 [WordOutput] {ChannellName = Enter name}
2 byte [Register] node 256, in %IB8.256 out %QB8.256 {ChannellName = 2 byte}
  STATUS_NASOS_1_VNUTR_2_SP_307 AT %QW8.256.0 [WordOutput] {ChannellName = Enter name}
2 byte [Register] node 257, in %IB8.257 out %QB8.257 {ChannellName = 2 byte}
  STATUS_NASOS_2_VNUTR_2_SP_307 AT %QW8.257.0 [WordOutput] {ChannellName = Enter name}
  STATUS_TRUBA_VNUTR_SP_307 AT %QW8.258.0 [WordOutput] {ChannellName = Enter name}
2 byte [Register] node 259, in %IB8.259 out %QB8.259 {ChannellName = 2 byte}
  AT %QW8.259.0 [WordOutput] {ChannellName = Enter name}
AT %QD9.0 [DWordOutput] Last address {ChannellName = Enter name}
ERROR_CONNECT AT %QW9.1 [WordOutput] Last error {ChannellName = Enter name}
Debug RS-232 [DEBUG_USART] node 0, in %IB9.0 out %QB9.0 {ChannellName = Debug RS-232; CommunicationSpeed = 115200; Parity = NO PARITY CHECK; BitLength = 8 bits; StopLength = One stop bit; InterfaceType = RS232; FrameOriented = ASCII; Timeout = 0; Visibility = No}
Universal Modbus device [ID2000] node 1, in %IB9.1 out %QB9.1 {ChannellName = Universal Modbus device; ModuleIP = 10:0:6:11; ServiceTimeout = 150; TCPport = 502; NetMode = TCP; ModuleSlaveAddress = 1; RequestType = Both; PeriodOfService = 50; Visibility = No; RepeatCounter = 0; ByteSequence = Native}
  AT %QB9.1.0 [ComChannel] Command (0xff - Start) {ChannellName = Enter name}
TEMPERATURA_1_PR_OTOPLENIYA_AI AT %QD9.1.0.0 [FloatOutput] {ChannellName = Enter name}
TEMPERATURA_2_OBR_OTOPLENIYA_AI AT %QD9.1.1.0 [FloatOutput] {ChannellName = Enter name}
TEMPERATURA_3_PR_GVS_AI AT %QD9.1.2.0 [FloatOutput] {ChannellName = Enter name}
TEMPERATURA_4_OBR_GVS_AI AT %QD9.1.3.0 [FloatOutput] {ChannellName = Enter name}
TEMPERATURA_5_KOTEL_1_AI AT %QD9.1.4.0 [FloatOutput] {ChannellName = Enter name}
TEMPERATURA_6_KOTEL_2_AI AT %QD9.1.5.0 [FloatOutput] {ChannellName = Enter name}
TEMPERATURA_7_KOTEL_3_AI AT %QD9.1.6.0 [FloatOutput] {ChannellName = Enter name}
TEMPERATURA_8_ULICA_AI AT %QD9.1.7.0 [FloatOutput] {ChannellName = Enter name}
Universal Modbus device [ID2000] node 2, in %IB9.2 out %QB9.2 {ChannellName = Universal Modbus device; ModuleIP = 10:0:6:12; ServiceTimeout = 150; TCPport = 502; NetMode = TCP; ModuleSlaveAddress = 1; RequestType = Both; PeriodOfService = 50; Visibility = No; RepeatCounter = 0; ByteSequence = Native}
  AT %QB9.2.0 [ComChannel] Command (0xff - Start) {ChannellName = Enter name}
DAVLENIE_1_PR_OTOPLENIYA_AI AT %QD9.2.0.0 [FloatOutput] {ChannellName = Enter name}
DAVLENIE_2_OBR_OTOPLENIYA_AI AT %QD9.2.1.0 [FloatOutput] {ChannellName = Enter name}
DAVLENIE_3_PR_GVS_AI AT %QD9.2.2.0 [FloatOutput] {ChannellName = Enter name}
DAVLENIE_4_OBR_GVS_AI AT %QD9.2.3.0 [FloatOutput] {ChannellName = Enter name}
DAVLENIE_5_PR_VNUTR_AI AT %QD9.2.4.0 [FloatOutput] {ChannellName = Enter name}
DAVLENIE_6_OBR_VNUTR_AI AT %QD9.2.5.0 [FloatOutput] {ChannellName = Enter name}
DAVLENIE_7_NAKOPITELNIY_BAK_AI AT %QD9.2.6.0 [FloatOutput] {ChannellName = Enter name}
AT %QD9.2.7.0 [FloatOutput] {ChannellName = Enter name}
Universal Modbus device [ID2000] node 3, in %IB9.3 out %QB9.3 {ChannellName = Universal Modbus device; ModuleIP = 10:0:6:14; ServiceTimeout = 150; TCPport = 502; NetMode = TCP; ModuleSlaveAddress = 1; RequestType = By poll time; PeriodOfService = 50; Visibility = No; RepeatCounter = 0; ByteSequence = Native}
  AT %QB9.3.0 [ComChannel] Command (0xff - Start) {ChannellName = Enter name}
xDO AT %QW9.3.0.0 [WordOutput] {ChannellName = Enter name}
RS-485-1 [COM1_USART] node 0, in %IB10.0 out %QB10.0 {ChannellName = RS-485-1; CommunicationSpeed = 9600; Parity = NO PARITY CHECK; BitLength = 8 bits; StopLength = One stop bit; InterfaceType = RS485; FrameOriented = ASCII; Timeout = 0; Visibility = No}
*)

(* POU PLC_PRG, ST *)
PROGRAM PLC_PRG
VAR
	I:INT;
	Tpr: REAL; (*-------------------------------------------------------------------------------------ДЛЯ ТЕМПЕРАТУРНОГО РЕЖИМА*)
	T_USTAVKA_T1: REAL;(*--------------------------------------------------------------------УСТАВКА ДЛЯ ПРЯМОЙ ОТОПЛЕНИЯ*)
	T_USTAVKA_T3: REAL;(*------------------------------------------------------------------------------УСТАВКА ДЛЯ ПРЯМОЙ ГВС*)
	PID_OTOPLENIE:PID_REGULATOR;(*---------------------------ПИД РЕГУЛИРОВАНИЕ СМЕСИТЕЛЬНОГО КРАНА ОТОПЛЕНИЕ*)
	PID_GVS:PID_REGULATOR;(*---------------------------------------------ПИД РЕГУЛИРОВАНИЕ СМЕСИТЕЛЬНОГО КРАНА ГВС*)
(*-----------------------------------------------------------------------------------------------------------------------------------------*)
	xDO0,(*---------------------------------------------------------------------------------------------------------НАСОС СЕТЕВОЙ 1*)
	xDO1,(*---------------------------------------------------------------------------------------------------------НАСОС СЕТЕВОЙ 2*)
	xDO2,(*----------------------------------------------------------------------------------------НАСОС ВНУТРЕННЕГО КОНТУРА 1*)
	xDO3,(*----------------------------------------------------------------------------------------НАСОС ВНУТРЕННЕГО КОНТУРА 2*)
	xDO4,(*---------------------------------------------------------------------------------------------------------------НАСОС ГВС 1*)
	xDO5,(*---------------------------------------------------------------------------------------------------------------НАСОС ГВС 2*)
	xDO6,(*--------------------------------------------------------------------------------------------------НАСОС ПОДПИТОЧНЫЙ 1*)
	xDO7,(*--------------------------------------------------------------------------------------------------НАСОС ПОДПИТОЧНЫЙ 2*)
	xDO8,(*----------------------------------------------------------------------------------------------НАСОС ЦИРКУЛЯЦИОННЫЙ 1*)
	xDO9, (*---------------------------------------------------------------------------------------------НАСОС ЦИРКУЛЯЦИОННЫЙ 2*)
	xDO10,(*--------------------------------------------------------------------------------------------НАСОС ЦИРКУЛЯЦИОННЫЙ 3*)
	xDO11,(*-------------------------------------------------------------------------------------------------ГОРЕЛКА 1: ТЕРМОСТАТ*)
	xDO12,(*-------------------------------------------------------------------------------------------------ГОРЕЛКА 2: ТЕРМОСТАТ*)
	xDO13,(*-------------------------------------------------------------------------------------------------ГОРЕЛКА 3: ТЕРМОСТАТ*)
	xDO14,(*------------------------------------------------------------*)
	xDO15:(*------------------------------------------------------------*)
																	   	    BOOL; (*---ЗНАЧЕНИЯ ДИСКРЕТНЫХ МОДУЛЕЙ МУ210-402*)
(*-----------------------------------------------------------------------------------------------------------------------------------------*)

(*-----------------------------------------------------------------------------------ПАРАМЕТРЫ ДЛЯ ВЫЧИСЛЕНИЯ ОШИБКИ МОДУЛЯ*)
	STEP_MODUL_ERROR:INT;
	TIMER_MODUL_ERROR:TP;
(*-----------------------------------------------------------------------------------------------------------------------------------------*)
	NARABOTKA_CHASOV:TON;(*---------------------------------------------------------ТАЙМЕР ДЛЯ НАРАБОТКИ ЧАСОВ/МИНУТ*)
(*---------------------------------------------------------------------------------------------------------ИНИЦИАЛИЗАЦИЯ НАСОСОВ*)



	STEP_ZIMNIY:INT;(*------------------------------------------------------------------------------------------------------------------------------------------УДАЛИТЬ*)
	STEP_LETNIY:INT;(*------------------------------------------------------------------------------------------------------------------------------------------УДАЛИТЬ*)

	KASKAD_NASOSOV_1_SETEVOY:KASKAD_2_NASOSA_2_DATCHIKA_DAVLENIA;
	PUSK_KASKAD_NASOSOV_1_SETEVOY:BOOL;
	WORK_KASKAD_1_SETEVOY:BOOL;(*-----------------------------------------------------------РАБОТА КАСКАДА 1 СЕТЕВОГО*)
	STEP_AVARIA_NIZKOE_DAVLENIE_SETEVOY:INT;
	TIMER_AVARIA_NIZKOE_DAVLENIE_SETEVOY:TP;

	KASKAD_NASOSOV_2_VNUTR:KASKAD_2_NASOSA_2_DATCHIKA_DAVLENIA;
	PUSK_KASKAD_NASOSOV_2_VNUTR:BOOL;
	WORK_KASKAD_2_VNUTR:BOOL;(*-----------------------------------------------------------РАБОТА КАСКАДА 2 ВНУТРЕННЕГО*)
	STEP_AVARIA_NIZKOE_DAVLENIE_VNUTR:INT;
	TIMER_AVARIA_NIZKOE_DAVLENIE_VNUTR:TP;

	KASKAD_NASOSOV_3_GVS:KASKAD_2_NASOSA_2_DATCHIKA_DAVLENIA;
	PUSK_KASKAD_NASOSOV_3_GVS:BOOL;
	WORK_KASKAD_3_GVS:BOOL;(*---------------------------------------------------------------------------РАБОТА КАСКАДА ГВС*)
	STEP_AVARIA_NIZKOE_DAVLENIE_GVS:INT;
	TIMER_AVARIA_NIZKOE_DAVLENIE_GVS:TP;

	KASKAD_NASOSOV_4_PODPITKA:KASKAD_PODPITKA_PO_DATCHIKU_OBRATKI;
	PUSK_KASKAD_NASOSOV_4_PODPITKA:BOOL;
	WORK_KASKAD_4_PODPITKA:BOOL;(*------------------------------------------------------------РАБОТА КАСКАДА ПОДПИТКА*)
	USTAVKA_DAVLENIA_PODPITKA:REAL;(*----------------------------УСТАВКА ОБРАТКИ ДЛЯ ПОДПИТКИ В ЗАВИСИМОСТИ ОТ
																			--------------------------ЗИМНЕГО ИЛИ ЛЕТНЕГО РЕЖИМА*)
(*----------------------------------------------------------------------------------------------------------ИНИЦИАЛИЗАЦИЯ ГОРЕЛОК*)
	GORELKA_1:GORELKA_ROSSEN;
	PUSK_GORELKA_1:BOOL;
	WORK_GORELKA_1:BOOL;(*-----------------------------------------------------------------------------------РАБОТА ГОРЕЛКИ 1*)
	STEP_STATUS_PREDUPREGDENIE_ON_GORELKA_1:INT;
	TIMER_STATUS_PREDUPREGDENIE_ON_GORELKA_1:TP;

	GORELKA_2:GORELKA_ROSSEN;
	PUSK_GORELKA_2:BOOL;
	WORK_GORELKA_2:BOOL;(*-----------------------------------------------------------------------------------РАБОТА ГОРЕЛКИ 2*)
	STEP_STATUS_PREDUPREGDENIE_ON_GORELKA_2:INT;
	TIMER_STATUS_PREDUPREGDENIE_ON_GORELKA_2:TP;

	GORELKA_3:GORELKA_ROSSEN;
	PUSK_GORELKA_3:BOOL;
	WORK_GORELKA_3:BOOL;(*-----------------------------------------------------------------------------------РАБОТА ГОРЕЛКИ 2*)
	STEP_STATUS_PREDUPREGDENIE_ON_GORELKA_3:INT;
	TIMER_STATUS_PREDUPREGDENIE_ON_GORELKA_3:TP;


	AVARIA_OSNOVNAYA_GORELKA:BOOL;
	AVARIA_SECOND_GORELKA:BOOL;
	AVARIA_RESERV_GORELKA:BOOL;

	STEP_PODOGREV_SECOND_GORELKA:INT;
	STEP_PODOGREV_RESERV_GORELKA:INT;
	STEP_AVARIA_PODOGREV_RESERV_GORELKA:INT;

(*----------------------------------------------------------------------------------------ИНИЦИАЛИЗАЦИЯ НАКОПИТЕЛЬНОГО БАКА*)
	BAK:NAKOPITELNYU_BAK;
(*-----------------------------------------------------------------------------------------------------------------------------------------*)

	R_TRIG1: R_TRIG;
	R_TRIG2: R_TRIG;
	R_TRIG3: R_TRIG;
	R_TRIG4: R_TRIG;
	R_TRIG5: R_TRIG;
	R_TRIG6: R_TRIG;
	R_TRIG7: R_TRIG;
	R_TRIG8: R_TRIG;
	R_TRIG9: R_TRIG;
	R_TRIG10: R_TRIG;
	R_TRIG11: R_TRIG;
	R_TRIG12: R_TRIG;
	R_TRIG13: R_TRIG;
	R_TRIG14: R_TRIG;

	DAVLENIE_1_ERROR: BYTE;
	DAVLENIE_2_ERROR: BYTE;
	DAVLENIE_3_ERROR: BYTE;
	DAVLENIE_4_ERROR: BYTE;
	DAVLENIE_5_ERROR: BYTE;
	DAVLENIE_6_ERROR: BYTE;
	DAVLENIE_7_ERROR: BYTE;

	TEMPERATURA_1_ERROR: BYTE;
	TEMPERATURA_2_ERROR: BYTE;
	TEMPERATURA_3_ERROR: BYTE;
	TEMPERATURA_4_ERROR: BYTE;
	TEMPERATURA_5_ERROR: BYTE;
	TEMPERATURA_6_ERROR: BYTE;
	TEMPERATURA_7_ERROR: BYTE;
	TEMPERATURA_8_ERROR: BYTE;

	DAVLENIE_1_DEC: DECODE_FLOAT;
	DAVLENIE_2_DEC: DECODE_FLOAT;
	DAVLENIE_3_DEC: DECODE_FLOAT;
	DAVLENIE_4_DEC: DECODE_FLOAT;
	DAVLENIE_5_DEC: DECODE_FLOAT;
	DAVLENIE_6_DEC: DECODE_FLOAT;
	DAVLENIE_7_DEC: DECODE_FLOAT;
	DAVLENIE_8_DEC: DECODE_FLOAT;

	TEMPERATURA_1_DEC: DECODE_FLOAT;
	TEMPERATURA_2_DEC: DECODE_FLOAT;
	TEMPERATURA_3_DEC: DECODE_FLOAT;
	TEMPERATURA_4_DEC: DECODE_FLOAT;
	TEMPERATURA_5_DEC: DECODE_FLOAT;
	TEMPERATURA_6_DEC: DECODE_FLOAT;
	TEMPERATURA_7_DEC: DECODE_FLOAT;
	TEMPERATURA_8_DEC: DECODE_FLOAT;

	OBRUV_DAVLENIYA_1: OBRYV_DATCHIKA;
	OBRUV_DAVLENIYA_2: OBRYV_DATCHIKA;
	OBRUV_DAVLENIYA_3: OBRYV_DATCHIKA;
	OBRUV_DAVLENIYA_4: OBRYV_DATCHIKA;
	OBRUV_DAVLENIYA_5: OBRYV_DATCHIKA;
	OBRUV_DAVLENIYA_6: OBRYV_DATCHIKA;
	OBRUV_DAVLENIYA_7: OBRYV_DATCHIKA;

	OBRUV_TEMPERATURU_1: OBRYV_DATCHIKA;
	OBRUV_TEMPERATURU_2: OBRYV_DATCHIKA;
	OBRUV_TEMPERATURU_3: OBRYV_DATCHIKA;
	OBRUV_TEMPERATURU_4: OBRYV_DATCHIKA;
	OBRUV_TEMPERATURU_5: OBRYV_DATCHIKA;
	OBRUV_TEMPERATURU_6: OBRYV_DATCHIKA;
	OBRUV_TEMPERATURU_7: OBRYV_DATCHIKA;
	OBRUV_TEMPERATURU_8: OBRYV_DATCHIKA;
(*-----------------------------------------------------------------------------------------------------------------------ОБРЫВ МОДУЛЯ*)
	KOLICHESTVO_OBRUV_MODUL:INT;
(*--------------------------------------------------------------------------------------------------ВСПОМОГАТЕЛЬНЫЙ ПЕРЕМЕННЫЕ*)
	DELTA_TEMPERATURA_USTAVKA:REAL;(*------------РАЗНИЦА МЕЖДУ УСТАВКОЙ И ТЕМПЕРАТУРОЙ ВЫХОДА ОТОПЛЕНИЯ*)
(*--------------------------------------------------------------------------------------------------------------------STEP ОБЪЯВЛЕНИЯ*)
	STEP_MAIN:INT;(*-------------------------------------------------------------------------------------ГЛАВНЫЙ ШАГ АЛГОРИТМА*)
	STEP_DAVL_POKOYA:INT;(*----------------------------------------ДЛЯ ПОДПИТКИ ПЕРЕД ВКЛЮЧЕНИЕМ СЕТЕВЫХ НАСОСОВ*)
	STEP_KASKAD_GVS:INT;(*--------------------------------------------------------------------------------------ДЛЯ ЗАПУСКА ГВС*)
	STEP_KASKAD_GORELKI:INT;(*--------------------------------------------------------------------------ДЛЯ КАСКАДА ГОРЕЛОК*)
	STEP_PODOGREV_2_GORELKOY:INT;(*---------------------------------------------------ДЛЯ ПОДОГРЕВА ВТОРОЙ ГОРЕЛКОЙ*)
	STEP3:INT;(*-------------------------------------------------------------------------ДЛЯ ПЕРЕКЛЮЧЕНИЯ ОСНОВНОЙ ГОРЕЛКИ*)
	STEP4:INT;(*-------------------------------------------------------------------------ДЛЯ ПЕРЕКЛЮЧЕНИЯ ОСНОВНОЙ ГОРЕЛКИ*)
	STEP_CIRCULAYCIONNUY_NASOS_1:INT;(*-----------------------------------ДЛЯ ОТКЛЮЧЕНИЯ ЦИРКУЛЯЦИОННОГО НАСОСА*)
	STEP_CIRCULAYCIONNUY_NASOS_2:INT;(*-----------------------------------ДЛЯ ОТКЛЮЧЕНИЯ ЦИРКУЛЯЦИОННОГО НАСОСА*)
	STEP_CIRCULAYCIONNUY_NASOS_3:INT;(*-----------------------------------ДЛЯ ОТКЛЮЧЕНИЯ ЦИРКУЛЯЦИОННОГО НАСОСА*)
	TIMER_CIRCUL_NASOS_1:TP;
	TIMER_CIRCUL_NASOS_2:TP;
	TIMER_CIRCUL_NASOS_3:TP;
	STEP_PODPITKA_OTOPLENIYA:INT;
	STEP_SBROS_OTOPLENIYA:INT;
	STEP_SBROS_GVS:INT;
	STEP_NAK_BAK:INT;(*-----------------------------------------------------------------------------ДЛЯ НАКОПИТЕЛЬНОГО БАКА*)
END_VAR
VAR RETAIN
(*--------------------------------------------------------------------------------------------------------------------------------АВАРИИ*)
(*'ЭТИ АВАРИИ НУЖНО ОБЪЯВИТЬ ВНУТРИ ПРОГРАММЫ *)
	AVARIA_OBRUV_DATCHIKA_TEMPERATURA_1_PR_OTOP:BOOL;(*-------АВАРИЯ ОБРЫВ ДАТЧИКА Т1 ПРЯМАЯ ОТОПЛЕНИЯ*)
	AVARIA_OBRUV_DATCHIKA_TEMPERATURA_2_OBR_OTOP:BOOL;(*---АВАРИЯ ОБРЫВ ДАТЧИКА Т2 ОБРАТКА ОТОПЛЕНИЯ*)
	AVARIA_OBRUV_DATCHIKA_TEMPERATURA_3_PR_GVS:BOOL;(*------------------АВАРИЯ ОБРЫВ ДАТЧИКА Т3 ПРЯМАЯ ГВС*)
	AVARIA_OBRUV_DATCHIKA_TEMPERATURA_4_OBR_GVS:BOOL;(*---------------АВАРИЯ ОБРЫВ ДАТЧИКА Т4 ОБРАТКА ГВС*)
	AVARIA_OBRUV_DATCHIKA_TEMPERATURA_5_KOTEL_1:BOOL;(*----------------------АВАРИЯ ОБРЫВ ДАТЧИКА Т5 КОТЕЛ 1*)
	AVARIA_OBRUV_DATCHIKA_TEMPERATURA_6_KOTEL_2:BOOL;(*----------------------АВАРИЯ ОБРЫВ ДАТЧИКА Т6 КОТЕЛ 2*)
	AVARIA_OBRUV_DATCHIKA_TEMPERATURA_7_KOTEL_3:BOOL;(*----------------------АВАРИЯ ОБРЫВ ДАТЧИКА Т7 КОТЕЛ 3*)
	AVARIA_OBRUV_DATCHIKA_TEMPERATURA_8_ULICA:BOOL;(*--------------------------АВАРИЯ ОБРЫВ ДАТЧИКА Т7 УЛИЦА*)

	AVARIA_OBRUV_DATCHIKA_DAVLENIE_1_PR_OTOP:BOOL;(*-----------АВАРИЯ ОБРЫВ ДАТЧИКА Р1 ПРЯМАЯ ОТОПЛЕНИЯ*)
	AVARIA_OBRUV_DATCHIKA_DAVLENIE_2_OBR_OTOP:BOOL;(*--------АВАРИЯ ОБРЫВ ДАТЧИКА Р2 ОБРАТКА ОТОПЛЕНИЯ*)
	AVARIA_OBRUV_DATCHIKA_DAVLENIE_3_PR_GVS:BOOL;(*-----------------------АВАРИЯ ОБРЫВ ДАТЧИКА Р3 ПРЯМАЯ ГВС*)
	AVARIA_OBRUV_DATCHIKA_DAVLENIE_4_OBR_GVS:BOOL;(*--------------------АВАРИЯ ОБРЫВ ДАТЧИКА Р4 ОБРАТКА ГВС*)
	AVARIA_OBRUV_DATCHIKA_DAVLENIE_5_PR_VNUTR:BOOL;(*-------------------АВАРИЯ ОБРЫВ ДАТЧИКА Р3 ПРЯМАЯ ВНУТ*)
	AVARIA_OBRUV_DATCHIKA_DAVLENIE_6_OBR_VNUTR:BOOL;(*--------------АВАРИЯ ОБРЫВ ДАТЧИКА Р4 ОБРАТКА ОБРАТ*)
	AVARIA_OBRUV_DATCHIKA_DAVLENIE_7_NAK_BAK:BOOL;(*--------------------------АВАРИЯ ОБРЫВ ДАТЧИКА Р5 НАК.БАК*)

	AVARIA_SETEVOY_NASOS_1:BOOL;(*--------------------------------------------------------------АВАРИЯ СЕТЕВОЙ НАСОС 1*)
	AVARIA_SETEVOY_NASOS_2:BOOL;(*--------------------------------------------------------------АВАРИЯ СЕТЕВОЙ НАСОС 2*)

	AVARIA_VNUTR_NASOS_1:BOOL;(*---------------------------------------------------------------------АВАРИЯ ВНУТР НАСОС 1*)
	AVARIA_VNUTR_NASOS_2:BOOL;(*---------------------------------------------------------------------АВАРИЯ ВНУТР НАСОС 2*)

	AVARIA_GVS_NASOS_1:BOOL;(*---------------------------------------------------------------------------АВАРИЯ НАСОС ГВС 1*)
	AVARIA_GVS_NASOS_2:BOOL;(*---------------------------------------------------------------------------АВАРИЯ НАСОС ГВС 2*)

	AVARIA_PODPITOCHNYU_NASOS_1:BOOL;(*------------------------------------------------АВАРИЯ ПОДПИТОЧНЫЙ НАСОС 1*)
	AVARIA_PODPITOCHNYU_NASOS_2:BOOL;(*------------------------------------------------АВАРИЯ ПОДПИТОЧНЫЙ НАСОС 2*)

	AVARIA_GORELKA_1:BOOL;(*---------------------------------------------------------------------------------АВАРИЯ ГОРЕЛКА 1*)
	AVARIA_GORELKA_2:BOOL;(*---------------------------------------------------------------------------------АВАРИЯ ГОРЕЛКА 2*)
	AVARIA_GORELKA_3:BOOL;(*---------------------------------------------------------------------------------АВАРИЯ ГОРЕЛКА 2*)


END_VAR
VAR (* helpers for the ST form of the networks *)
	_t5 : TIME;
END_VAR
IF BIT_VKLUCHENIYA_SP_307=TRUE THEN (*-----------------------------------------------------------------------БИТ ВКЛЮЧЕНИЯ*)
(*---------------------------------------------------------------------------------------------------------------------------------МОДЕМ*)

MODEM;

(*----------------------------------------------------------------------------------------------------ДИСКРЕТНЫЙ ВЫВОД НА МОДУЛЬ*)
DO_DISKRETNUY_OUT;
(*---------------------------------------------------------------------------------------------------------------------ОБРЫВ ДАТЧИКОВ*)
DECOD_ERROR;
IF PUSK_SP_307 THEN
	AVARIA_DATCHIK;(*---------------------ЧТО БЫ НЕ ЛЕТЕЛИ АВАРИИ ОБРЫВА ДАТЧИКОВ ПОКА КОТЕЛЬНАЯ НЕ ЗАПУЩЕНА*)
END_IF
(*-------------------------------------------------------------------------------------------------------------------НАРАБОТКА МИНУТ*)
NARABOTKA_MINUT;
(*------------------------------------------------------------------------------------------------------------------------ОТВАЛ МОДУЛЯ*)

MODUL_ERROR;

(*-------------------------------------------------------------------------------------------------------------НАРАБОТКА ВКЛЮЧЕНИЙ*)
NARABOTKA_VKLUCHENIY;
(*--------------------------------------------------------------------------------------------------------ПОГОДОЗАВИСИМЫЙ ГРАФИК*)
TEMPERATURNYU_REGIM;
(*----------------------------------------------------------------------------------------------------АЛГОРИТМ РАБОТЫ КОТЕЛЬНОЙ*)
ALGORITHM;

(*---------------------------------------------------------------------------------------------------------ЦИРКУЛЯЦИОННЫЙ НАСОСЫ*)
CIRCULAYCIONNYE_NASOSU;
(*-------------------------------------------------------------------------------------------------------КАСКАД НАСОСОВ 1 СЕТЕВОЙ*)
KASKAD_NASOSOV_1_SETEVOY(
	OSNOVNOY:=REAL_TO_INT(OSNOVNOY_SETEVOY_NASOS),(*---------------------------------------------ОСНОВНОЙ НАСОС*)
	TIME_AVARIA:=REAL_TO_TIME(AVAR_VREMA_NASOS_OTOPL*1000),(*-----------------------------------ВРЕМЯ НА АВАРИЮ*)
	P_1:=DAVLENIE_1_PR_OTOPLENIYA_AI_SP_307,(*------------------------------------------------ДАВЛЕНИЕ ПОСЛЕ КАСКАДА*)
	P_2:=DAVLENIE_2_OBR_OTOPLENIYA_AI_SP_307, (*--------------------------------------------ДАВЛЕНИЕ ПЕРЕД КАСКАДОМ*)
	PEREPAD_DAVLENIA:=PEREPAD_DAVL_OTOP, (*-----------------------------------------------------------ПЕРЕПАД ДАВЛЕНИЯ*)
	SBROS_ERROR:=SBROS_AVARIA_SETEVOY_KASKAD_1_SP_307, (*---------------------СБРОС ОШИБКИ КАСКАДА НАСОСОВ*)
	PUSK_NASOS:=PUSK_KASKAD_NASOSOV_1_SETEVOY, (*------------------------------------------ПУСК КАСКАДА НАСОСОВ*)
	ERROR_NASOS1:=AVARIA_SETEVOY_NASOS_1, (*----------------ОШИБКА НАСОСА 1. ХРАНИТСЯ В RETAIN КОНТРОЛЛЕРА*)
	ERROR_NASOS2:=AVARIA_SETEVOY_NASOS_2, (*----------------ОШИБКА НАСОСА 2. ХРАНИТСЯ В RETAIN КОНТРОЛЛЕРА*)
	RELE_NASOS1=>xDO0, (*---------------------------------------------------------------------------РЕЛЕ ВКЛЮЧЕНИЯ НАСОСА 1*)
	RELE_NASOS2=>xDO1, (*---------------------------------------------------------------------------РЕЛЕ ВКЛЮЧЕНИЯ НАСОСА 2*)
	WORK=>WORK_KASKAD_1_SETEVOY,(*--------------------------------------------------СТАТУС РАБОТА КАСКАДА НАСОСОВ*)
);
(*--------------------------------------------------------------------------------------------------------КАСКАД НАСОСОВ 2 ЛЕТНИЙ*)
KASKAD_NASOSOV_2_VNUTR(
	OSNOVNOY:=REAL_TO_INT(OSNOVNOY_VNUTR_NASOS),(*---------------------------------------------ОСНОВНОЙ НАСОС*)
	TIME_AVARIA:=REAL_TO_TIME(AVAR_VREMA_NASOS_VNUTR*1000),(*-----------------------------------ВРЕМЯ НА АВАРИЮ*)
	P_1:=DAVLENIE_5_PR_VNUTR_AI_SP_307,(*------------------------------------------------ДАВЛЕНИЕ ПОСЛЕ КАСКАДА*)
	P_2:=DAVLENIE_6_OBR_VNUTR_AI_SP_307, (*--------------------------------------------ДАВЛЕНИЕ ПЕРЕД КАСКАДОМ*)
	PEREPAD_DAVLENIA:=PEREPAD_DAVL_VNUTR, (*-----------------------------------------------------------ПЕРЕПАД ДАВЛЕНИЯ*)
	SBROS_ERROR:=SBROS_AVARIA_VNUTR_KASKAD_2_SP_307, (*---------------------СБРОС ОШИБКИ КАСКАДА НАСОСОВ*)
	PUSK_NASOS:=PUSK_KASKAD_NASOSOV_2_VNUTR, (*------------------------------------------ПУСК КАСКАДА НАСОСОВ*)
	ERROR_NASOS1:=AVARIA_VNUTR_NASOS_1, (*----------------ОШИБКА НАСОСА 1. ХРАНИТСЯ В RETAIN КОНТРОЛЛЕРА*)
	ERROR_NASOS2:=AVARIA_VNUTR_NASOS_2, (*----------------ОШИБКА НАСОСА 2. ХРАНИТСЯ В RETAIN КОНТРОЛЛЕРА*)
	RELE_NASOS1=>xDO2, (*---------------------------------------------------------------------------РЕЛЕ ВКЛЮЧЕНИЯ НАСОСА 1*)
	RELE_NASOS2=>xDO3, (*---------------------------------------------------------------------------РЕЛЕ ВКЛЮЧЕНИЯ НАСОСА 2*)
	WORK=>WORK_KASKAD_2_VNUTR,(*--------------------------------------------------СТАТУС РАБОТА КАСКАДА НАСОСОВ*)
);
(*-------------------------------------------------------------------------------------------------------------КАСКАД НАСОСОВ 3 ГВС*)
KASKAD_NASOSOV_3_GVS(
	OSNOVNOY:=REAL_TO_INT(OSNOVNOY_GVS_NASOS),(*---------------------------------------------------ОСНОВНОЙ НАСОС*)
	TIME_AVARIA:=REAL_TO_TIME(AVAR_VREMA_NASOS_GVS*1000),(*--------------------------------------ВРЕМЯ НА АВАРИЮ*)
	P_1:=DAVLENIE_3_PR_GVS_AI_SP_307,(*----------------------------------------------------------ДАВЛЕНИЕ ПОСЛЕ КАСКАДА*)
	P_2:=DAVLENIE_4_OBR_GVS_AI_SP_307, (*------------------------------------------------------ДАВЛЕНИЕ ПЕРЕД КАСКАДОМ*)
	PEREPAD_DAVLENIA:=PEREPAD_DAVL_GVS, (*-------------------------------------------------------------ПЕРЕПАД ДАВЛЕНИЯ*)
	SBROS_ERROR:=SBROS_AVARIA_GVS_KASKAD_3_SP_307, (*---------------------------СБРОС ОШИБКИ КАСКАДА НАСОСОВ*)
	PUSK_NASOS:=PUSK_KASKAD_NASOSOV_3_GVS, (*-------------------------------------------------ПУСК КАСКАДА НАСОСОВ*)
	ERROR_NASOS1:=AVARIA_GVS_NASOS_1, (*----------------------ОШИБКА НАСОСА 1. ХРАНИТСЯ В RETAIN КОНТРОЛЛЕРА*)
	ERROR_NASOS2:=AVARIA_GVS_NASOS_2, (*----------------------ОШИБКА НАСОСА 2. ХРАНИТСЯ В RETAIN КОНТРОЛЛЕРА*)
	RELE_NASOS1=>xDO4, (*---------------------------------------------------------------------------РЕЛЕ ВКЛЮЧЕНИЯ НАСОСА 1*)
	RELE_NASOS2=>xDO5, (*---------------------------------------------------------------------------РЕЛЕ ВКЛЮЧЕНИЯ НАСОСА 2*)
	WORK=>WORK_KASKAD_3_GVS(*---------------------------------------------------------СТАТУС РАБОТА КАСКАДА НАСОСОВ*)
);
(*----------------------------------------------------------------------------------------------КАСКАД ПОДПИТОЧНЫЙХ НАСОСОВ 4*)
(*------В ЗАВИСИМОСТИ ОТ ТОГО В КАКОМ РЕЖИМЕ РАБОТАЕТ КОТЕЛЬНАЯ (ЗИМНИЙ ИЛИ ЛЕТНИЙ) БЕРЕТСЯ УСТАВКА ДЛЯ *)
(*-------------------------------------------------------------------------------ПОДПИТКИ ОТ КОТОРОЙ ОТСЧИТЫВАЕТСЯ АВАРИЯ*)

USTAVKA_DAVLENIA_PODPITKA:=USTAVKA_DAVL_OBR_OTOP_ZIMNIY;(*----------------------------------УСТАВКА ПОДПИТКИ*)

(*IF LETNIY_KASKAD_PUSK_SP_307 THEN USTAVKA_DAVLENIA_PODPITKA:=USTAVKA_DAVL_OBR_LETNIY; END_IF ----------------------------------------------------------------УДАЛИТЬ*)

KASKAD_NASOSOV_4_PODPITKA(
	OSNOVNOY:=REAL_TO_INT(OSNOVNOY_PODPITOCHNIY_NASOS),(*-------------------------------------ОСНОВНОЙ НАСОС*)
	TIME_AVARIA:=REAL_TO_TIME(AVAR_VREMA_NASOS_PODPITKI*1000),(*-------------------------------ВРЕМЯ НА АВАРИЮ*)
	P:=DAVLENIE_2_OBR_OTOPLENIYA_AI_SP_307,(*-----------------------ДАВЛЕНИЕ ОБРАТКИ ПОДПИТЫВАЕМОГО КОНТУРА*)
	USTAVKA_P:=USTAVKA_DAVLENIA_PODPITKA, (*-----------------------------------------------------------УСТАВКА ОБРАТКИ*)(*<------------------------------------------ ВОТ ЭТОТ ПАРАМЕТР НУЖНО НА ЗИМНИЙ И ЛЕТНИЙ РАЗВЕСТИ, ДАВЛЕНИЯ БУДУТ РАЗНЫЕ*)
	SBROS_ERROR:=SBROS_AVARIA_PODPITOCHNY_KASKAD_4_SP_307, (*---------------СБРОС ОШИБКИ КАСКАДА НАСОСОВ*) (*--------------------------------------------ДОБАВИЛ , НАДО ПРОВЕРЯТЬ*)
	PUSK_NASOS:=PUSK_KASKAD_NASOSOV_4_PODPITKA, (*------------------------------------------ПУСК КАСКАДА НАСОСОВ*)
	ERROR_NASOS1:=AVARIA_PODPITOCHNYU_NASOS_1, (*---------ОШИБКА НАСОСА 1. ХРАНИТСЯ В RETAIN КОНТРОЛЛЕРА*)
	ERROR_NASOS2:=AVARIA_PODPITOCHNYU_NASOS_2, (*---------ОШИБКА НАСОСА 2. ХРАНИТСЯ В RETAIN КОНТРОЛЛЕРА*)
	RELE_NASOS1=>xDO6, (*---------------------------------------------------------------------------РЕЛЕ ВКЛЮЧЕНИЯ НАСОСА 1*)
	RELE_NASOS2=>xDO7, (*---------------------------------------------------------------------------РЕЛЕ ВКЛЮЧЕНИЯ НАСОСА 2*)
	WORK=>WORK_KASKAD_4_PODPITKA,(*-------------------------------------------------СТАТУС РАБОТА КАСКАДА НАСОСОВ*)
);
(*------------------------------------------------------------------------------------------------ТРЕХХОДОВОЙ КРАН ОТОПЛЕНИЕ  1*)
IF PUSK_ESBE_SP_307 THEN
PID_OTOPLENIE(
	USTAVKA:=T_USTAVKA_T1,
	KORREKTIROVKA:=KORREKTIROVKA_USTAVKI_ESBE_1,
	SBROS:=SBROS_ESBE_1_SP_307,
	TEMPERATURA_IN:=TEMPERATURA_1_PR_OTOPLENIYA_AI_SP_307,
	ESBE_VREMYA_HODA_ZADVIGKI:=VREMYA_HODA_ZADVIZKI_ESBE_1,
	ESBE_MIN_VREMYA_HODA:=MIN_VREMYA_HODA_ESBE_1,
	ESBE_MIN_VREMYA_OSTANOVKI:=MIN_VREMYA_OSTANOVKI_ESBE_1,
	ESBE_PROPORCIONAL:=PROPORCIONALNAYA_SOSTAV_ESBE_1,
	ESBE_INTEGRAL:=INTEGRALNAYA_SOSTAV_ESBE_1,
	ESBE_DIFFERINCAL:=DIFFERENCIALNAYA_SOSTAV_ESBE_1,
	LESS=>ESBE_1_LESS,
	MORE=>ESBE_1_MORE,
);
END_IF
(*----------------------------------------------------------------------------------------------------------ТРЕХХОДОВОЙ КРАН ГВС  2*)
T_USTAVKA_T3:=USTAVKA_POSTOYANNAYA_ESBE_2+KORREKTIROVKA_USTAVKI_ESBE_2;
IF PUSK_ESBE_SP_307 THEN
PID_GVS(
	USTAVKA:=USTAVKA_POSTOYANNAYA_ESBE_2,
	KORREKTIROVKA:=KORREKTIROVKA_USTAVKI_ESBE_2,
	SBROS:=SBROS_ESBE_2_SP_307,
	TEMPERATURA_IN:=TEMPERATURA_3_PR_GVS_AI_SP_307,
	ESBE_VREMYA_HODA_ZADVIGKI:=VREMYA_HODA_ZADVIZKI_ESBE_2,
	ESBE_MIN_VREMYA_HODA:=MIN_VREMYA_HODA_ESBE_2,
	ESBE_MIN_VREMYA_OSTANOVKI:=MIN_VREMYA_OSTANOVKI_ESBE_2,
	ESBE_PROPORCIONAL:=PROPORCIONALNAYA_SOSTAV_ESBE_2,
	ESBE_INTEGRAL:=INTEGRALNAYA_SOSTAV_ESBE_2,
	ESBE_DIFFERINCAL:=DIFFERENCIALNAYA_SOSTAV_ESBE_2,
	LESS=>ESBE_2_LESS,
	MORE=>ESBE_2_MORE,
);
END_IF
(*-----------------------------------------------------------------------------------------------------------------------------ГОРЕЛКА 1*)
GORELKA_1(
	PUSK:=PUSK_GORELKA_1,
	TEMPERATURA_KOTLA:=TEMPERATURA_5_KOTEL_1_AI_SP_307,
	AVARIA:=S3_GORELKA_1,(*---------------------------------------------------------------------------------ОШИБКА С ГОРЕЛКИ 220 В*)
	AVAR_TEMPERATURA:=TEMPERATURA_AVARIA_MAX_GORELKA_1,
	SBROS_ERROR:=SBROS_AVARIA_GORELKA_1_SP_307,(*---------------------------------------------СБРОС АВАРИИ ГОРЕЛКИ*)
	ERROR_GORELKA:=AVARIA_GORELKA_1,(*------------------------------------------------------------------------------АВАРИЯ ГОРЕЛКА 1*)
	TERM=>xDO11,(*----------------------------------------------------------------------------------КЛЕММЫ ЗАПРОС НА РОЗЖИГ*)
	WORK=>WORK_GORELKA_1,(*-------------------------------------------------------------------------СТАТУС РАБОТА ГОРЕЛКИ*)
);
(*----------------------------------------------------------------------------------------------------------------------------ГОРЕЛКА 2*)
GORELKA_2(
	PUSK:=PUSK_GORELKA_2,
	TEMPERATURA_KOTLA:=TEMPERATURA_6_KOTEL_2_AI_SP_307,
	AVARIA:=S3_GORELKA_2,(*---------------------------------------------------------------------------------ОШИБКА С ГОРЕЛКИ 220 В*)
	AVAR_TEMPERATURA:=TEMPERATURA_AVARIA_MAX_GORELKA_2,
	SBROS_ERROR:=SBROS_AVARIA_GORELKA_2_SP_307,(*---------------------------------------------СБРОС АВАРИИ ГОРЕЛКИ*)
	ERROR_GORELKA:=AVARIA_GORELKA_2,(*------------------------------------------------------------------------------АВАРИЯ ГОРЕЛКА 1*)
	TERM=>xDO12,(*----------------------------------------------------------------------------------КЛЕММЫ ЗАПРОС НА РОЗЖИГ*)
	WORK=>WORK_GORELKA_2,(*-------------------------------------------------------------------------СТАТУС РАБОТА ГОРЕЛКИ*)
);
(*----------------------------------------------------------------------------------------------------------------------------ГОРЕЛКА 3*)
GORELKA_3(
	PUSK:=PUSK_GORELKA_3,
	TEMPERATURA_KOTLA:=TEMPERATURA_7_KOTEL_3_AI_SP_307,
	AVARIA:=S3_GORELKA_3,(*---------------------------------------------------------------------------------ОШИБКА С ГОРЕЛКИ 220 В*)
	AVAR_TEMPERATURA:=TEMPERATURA_AVARIA_MAX_GORELKA_3,
	SBROS_ERROR:=SBROS_AVARIA_GORELKA_3_SP_307,(*---------------------------------------------СБРОС АВАРИИ ГОРЕЛКИ*)
	ERROR_GORELKA:=AVARIA_GORELKA_3,(*------------------------------------------------------------------------------АВАРИЯ ГОРЕЛКА 1*)
	TERM=>xDO13,(*----------------------------------------------------------------------------------КЛЕММЫ ЗАПРОС НА РОЗЖИГ*)
	WORK=>WORK_GORELKA_3,(*-------------------------------------------------------------------------СТАТУС РАБОТА ГОРЕЛКИ*)
);
(*----------------------------------------------------------------------------------------------------------------НАКОПИТЕЛЬНЫЙ БАК*)
BAK(
	P:=DAVLENIE_7_NAKOPITELNIY_BAK_AI_SP_307,(*--------------------------ДАВЛЕНИЕ ДАТЧИКА НАКОПИТЕЛЬНОГО БАКА*)
	D_MIN:=BAK_NIGNAYA_GRANICA,(*-----------------------------------------------------------ДАВЛЕНИЕ МИНИМАЛЬНОЕ В 0%*)
	D_MAX:=BAK_VERHNYAY_GRANICA,(*-----------------------------------------------------ДАВЛЕНИЕ МАКСИМАЛЬНОЕ В 100%*)
	PROCENT_ZAPOLNENIA=>STATUS_BAK_PROCENT_ZAPOLNENIA, (*----------------------------------ПРОЦЕНТ ЗАПОЛНЕНИЯ*)
);
(*-----------------------------------------------------------------------------------------------------------------------------------------*)

(*----СБРОС ОШИБОК ДОЛЖЕН ВЫПОЛНЯТЬСЯ В САМОМ КОНЦЕ ПОСЛЕ ИНИЦИАЛИЗАЦИЙ ВСЕХ ФУНКЦИОНАЛЬНЫХ БЛОКОВ*)
(*-----------------------------------------------------------------------------------------------------------------ОБРАБОТКА АВАРИЙ*)

IF PUSK_SP_307 THEN
	AVARIA_STATUS;
END_IF

(*-----------------------------------------------------------------------------------------------------------------ОБРАБОТКА АВАРИЙ*)

OBRABOTKA_AVARIY;

(*-----------------------------------------------------------------------------------------------------------------------СБРОС ОШИБОК*)

SBROS_ERROR;
(*-----------------------------------------------------------------------------------СТАТУСЫ ЭЛЕМЕНТОВ КОТЕЛЬНОЙ ДЛЯ ПАНЕЛИ*)
OUT_STATUS_SP_307;
END_IF (*--------------------------------------------------------------------------------------------------------------БИТ ВКЛЮЧЕНИЯ*)
END_PROGRAM
ACTION ALGORITHM:
(*----------------------------------------------------------------------------------------------------------------НАКОПИТЕЛЬНЫЙ БАК*)
IF STATUS_BAK_PROCENT_ZAPOLNENIA<BAK_USTAVKA_NAPOLNENIA AND STEP_NAK_BAK=0  THEN
	STEP_NAK_BAK:=1;
END_IF
CASE STEP_NAK_BAK OF
	1:
		EL_KL_4_NAK_BAK:=TRUE; (*-------------------------------------------------------------ВКЛЮЧАЕМ КЛАПАН НАКОПИТЕЛЬНОГО БАКА*)
		IF STATUS_BAK_PROCENT_ZAPOLNENIA>=BAK_USTAVKA_NAPOLNENIA+BAK_GISTEREZIS_NAPOLNENIA THEN
			STEP_NAK_BAK:=2;
		END_IF
	2:
		EL_KL_4_NAK_BAK:=FALSE; (*-----------------------------------------------------------ОТКЛЮЧАЕМ КЛАПАН НАКОПИТЕЛЬНОГО БАКА*)
		STEP_NAK_BAK:=0;
END_CASE





(*------------------------------------------------------------------РАСЧЕТ ОТКЛОНЕНИЯ ТЕМПЕРАТУРЫ ОТОПЛЕНИЯ ОТ УСТАВКИ*)
DELTA_TEMPERATURA_USTAVKA:=T_USTAVKA_T1-TEMPERATURA_1_PR_OTOPLENIYA_AI_SP_307;
(*-----------------------------------------------------------------------------------------------------------------------------------------*)



(*------------------------ЕСЛИ ПУСК КОТЕЛЬНАЯ НАЖАТА  И МОДУЛИ НЕ ОТВАЛИЛИСЬ ТО НАЧИНАЕМ ВЫПОЛНЯТЬ АЛГОРИТМ*)
(*----------------------------------------------------------------------------------------------------------------ЗАПУСК НАСОСОВ ГВС*)
IF PUSK_SP_307=TRUE AND ERROR_MODUL_SP_307=FALSE AND AVARIA_PHASA_SP_307=FALSE AND PUSK_GVS_SP_307
AND AVARIA_VUSOKOE_DAVLENIE_GVS_SP_307=FALSE AND AVARIA_NIZKOE_DAVLENIE_GVS_SP_307=FALSE AND AVARIA_FIRE_SP_307=FALSE AND AVARIA_GAZ_SP_307=FALSE  THEN
	IF AVARIA_GVS_NASOS_1=FALSE OR AVARIA_GVS_NASOS_2=FALSE THEN
		PUSK_KASKAD_NASOSOV_3_GVS:=TRUE;
	ELSE
		PUSK_KASKAD_NASOSOV_3_GVS:=FALSE;
	END_IF
ELSE
	PUSK_KASKAD_NASOSOV_3_GVS:=FALSE;
	xDO.4:=xDO4:=FALSE;(*---------------------------------------------------------------------------------------------НАСОС ГВС 1*)
	xDO.5:=xDO5:=FALSE;(*---------------------------------------------------------------------------------------------НАСОС ГВС 2*)
END_IF


IF PUSK_SP_307=TRUE AND ERROR_MODUL_SP_307=FALSE AND AVARIA_PHASA_SP_307=FALSE AND VNUTR_KASKAD_PUSK_SP_307
(*AND AVARIA_VUSOKOE_DAVLENIE_OTOPLENIYA_SP_307=FALSE AND AVARIA_NIZKOE_DAVLENIE_OTOPLENIYA_SP_307=FALSE AND STEP_MAIN>101*)  THEN
	IF AVARIA_VNUTR_NASOS_1=FALSE OR AVARIA_VNUTR_NASOS_2=FALSE  THEN
		PUSK_KASKAD_NASOSOV_2_VNUTR:=TRUE;
	ELSE
		PUSK_KASKAD_NASOSOV_2_VNUTR:=FALSE;
	END_IF
ELSE
	PUSK_KASKAD_NASOSOV_2_VNUTR:=FALSE;
	xDO.2:=xDO2:=FALSE;(*-------------------------------------------------------------------------------НАСОС ВНУТР.КОНТУРА 1*)
	xDO.3:=xDO3:=FALSE;(*-------------------------------------------------------------------------------НАСОС ВНУТР.КОНТУРА 2*)
END_IF

(*--------------------------------------------------------------------------------------------------------------СБРОС ОТОПЛЕНИЯ*)
	IF DAVLENIE_1_PR_OTOPLENIYA_AI_SP_307>EL_2_DAVL_SBROSA_PR_OTOP
  	 AND STEP_SBROS_OTOPLENIYA=0 THEN
		STEP_SBROS_OTOPLENIYA:=1;
	END_IF
	CASE STEP_SBROS_OTOPLENIYA OF
		1:
			EL_KL_2_SBROS_OTOPL:=TRUE; (*-----------------------------------------------ВКЛЮЧЕНИЕ КЛАПАНА СБРОСА ОТОПЛЕНИ*)
			IF DAVLENIE_1_PR_OTOPLENIYA_AI_SP_307<=EL_2_DAVL_SBROSA_PR_OTOP-GISTEREZIS_SBROS_OTOPLENIYA THEN
				STEP_SBROS_OTOPLENIYA:=2;
			END_IF
		2:
			EL_KL_2_SBROS_OTOPL:=FALSE; (*----------------------------------------------ВЫКЛЮЧЕНИЕ КЛАПАНА СБРОСА ОТОПЛЕНИЯ*)
			STEP_SBROS_OTOPLENIYA:=0;
	END_CASE

(*--------------------------------------------------------------------------------------------------------------СБРОС ГВС*)
	IF DAVLENIE_3_PR_GVS_AI_SP_307>EL_3_DAVL_SBROSA_GVS
  	 AND STEP_SBROS_GVS=0 THEN
		STEP_SBROS_GVS:=1;
	END_IF
	CASE STEP_SBROS_GVS OF
		1:
			EL_KL_3_SBROS_GVS:=TRUE; (*-----------------------------------------------ВКЛЮЧЕНИЕ КЛАПАНА СБРОСА ОТОПЛЕНИ*)
			IF DAVLENIE_3_PR_GVS_AI_SP_307<=EL_3_DAVL_SBROSA_GVS-GISTEREZIS_SBROS_GVS THEN
				STEP_SBROS_GVS:=2;
			END_IF
		2:
			EL_KL_3_SBROS_GVS:=FALSE; (*----------------------------------------------ВЫКЛЮЧЕНИЕ КЛАПАНА СБРОСА ОТОПЛЕНИЯ*)
			STEP_SBROS_GVS:=0;
	END_CASE



(*--------------------------------------------------------------------------------------------------------------ПОДПИТКА ОТОПЛЕНИЯ*)
	IF DAVLENIE_2_OBR_OTOPLENIYA_AI_SP_307<USTAVKA_DAVL_OBR_OTOP_ZIMNIY AND WORK_KASKAD_1_SETEVOY
  	 AND STEP_PODPITKA_OTOPLENIYA=0
	AND (AVARIA_PODPITOCHNYU_NASOS_1=FALSE OR AVARIA_PODPITOCHNYU_NASOS_2=FALSE)THEN
		STEP_PODPITKA_OTOPLENIYA:=1;
	END_IF
	CASE STEP_PODPITKA_OTOPLENIYA OF
		1:
			EL_KL_1_PODPITKA_OTOPL:=TRUE; (*-----------------------------------------------ВКЛЮЧЕНИЕ КЛАПАНА ПОДПИТКИ*)
			PUSK_KASKAD_NASOSOV_4_PODPITKA:=TRUE;
			IF DAVLENIE_2_OBR_OTOPLENIYA_AI_SP_307>=USTAVKA_DAVL_OBR_OTOP_ZIMNIY+GISTEREZIS_PODPITKI_OTOPL THEN
				STEP_PODPITKA_OTOPLENIYA:=2;
			END_IF
			IF  AVARIA_PODPITOCHNYU_NASOS_1  AND AVARIA_PODPITOCHNYU_NASOS_2  THEN
				STEP_PODPITKA_OTOPLENIYA:=2;
			END_IF
			IF WORK_KASKAD_1_SETEVOY=FALSE OR (AVARIA_SETEVOY_NASOS_1
			AND AVARIA_SETEVOY_NASOS_2) THEN
				STEP_PODPITKA_OTOPLENIYA:=2;
			END_IF
		2:
			EL_KL_1_PODPITKA_OTOPL:=FALSE; (*----------------------------------------------ВКЛЮЧЕНИЕ КЛАПАНА ПОДПИТКИ*)
			PUSK_KASKAD_NASOSOV_4_PODPITKA:=FALSE;
			STEP_PODPITKA_OTOPLENIYA:=0;
	END_CASE




(*--------------------------------------------------------------------------------------------------------ЗАПУСК СЕТЕВОГО КОНТУРА*)
IF PUSK_SP_307=TRUE AND ERROR_MODUL_SP_307=FALSE AND AVARIA_PHASA_SP_307=FALSE
AND AVARIA_VUSOKOE_DAVLENIE_OTOPLENIYA_SP_307=FALSE
AND AVARIA_NIZKOE_DAVLENIE_OTOPLENIYA_SP_307=FALSE  THEN
	CASE STEP_MAIN OF
		0: 						(*-------------------------------------------------------------------------------------ВКЛЮЧЕНИЕ ГАЗА*)
			(*xDO11:=TRUE;*)(*--------------------------------------------------------------------------------------------------------------------------КЛАПАНА ГАЗА НЕТ*)
			STEP_MAIN:=100;
		100:	                   (*-------ПЕРВОНАЧАЛЬНАЯ ПОДПИТКА ПРЯМОЙ ОТОПЛЕНИЯ ПЕРЕД ЗАПУСКОМ СЕТЕВЫХ НАСОСОВ*)
			IF (DAVLENIE_1_PR_OTOPLENIYA_AI<DAVL_POKOYA_OTOP) AND FIRST_START_SP_307  THEN
				STEP_MAIN:=101;
				STEP_DAVL_POKOYA:=1;
			ELSE
				STEP_MAIN:=110;
				STEP_KASKAD_GVS:=10;
			END_IF
		101: (*----------------------------------------------------------------------ПОДПИТЫВАЕМ СЕТЕВОЙ КОНТУР ДО УСТАВКИ*)
			CASE STEP_DAVL_POKOYA OF
				1:
					IF DAVLENIE_1_PR_OTOPLENIYA_AI<DAVL_POKOYA_OTOP THEN
						EL_KL_1_PODPITKA_OTOPL:=TRUE;  (*--------------------------------ВКЛЮЧЕНИЕ ЭЛЕКТРОКЛАПАНА 1 ПОДПИТКИ ОТОПЛЕНИЯ*)
					END_IF
					STEP_DAVL_POKOYA:=2;
				2:
					PUSK_KASKAD_NASOSOV_4_PODPITKA:=TRUE;
					IF AVARIA_PODPITOCHNYU_NASOS_1 AND AVARIA_PODPITOCHNYU_NASOS_2 THEN
						STEP_DAVL_POKOYA:=4;
					END_IF
					IF DAVLENIE_1_PR_OTOPLENIYA_AI>DAVL_POKOYA_OTOP THEN
						EL_KL_1_PODPITKA_OTOPL:=FALSE;  (*-----------------------------ВЫКЛЮЧЕНИЕ ЭЛЕКТРОКЛАПАНА 1 ПОДПИТКИ ОТОПЛЕНИЯ*)
					ELSE
						EL_KL_1_PODPITKA_OTOPL:=TRUE;  (*--------------------------------ВКЛЮЧЕНИЕ ЭЛЕКТРОКЛАПАНА 1 ПОДПИТКИ ОТОПЛЕНИЯ*)
					END_IF

					IF DAVLENIE_1_PR_OTOPLENIYA_AI>DAVL_POKOYA_OTOP THEN
						STEP_DAVL_POKOYA:=3;
					END_IF
				3:
					PUSK_KASKAD_NASOSOV_4_PODPITKA:=FALSE;
					EL_KL_1_PODPITKA_OTOPL:=FALSE;  (*---------------------------------ВЫКЛЮЧЕНИЕ ЭЛЕКТРОКЛАПАНА 1 ПОДПИТКИ ОТОПЛЕНИЯ*)
					STEP_MAIN:=110;
					STEP_KASKAD_GVS:=10;
					STEP_DAVL_POKOYA:=0;
				4:
					PUSK_KASKAD_NASOSOV_4_PODPITKA:=FALSE;
					EL_KL_1_PODPITKA_OTOPL:=FALSE;  (*---------------------------------ВЫКЛЮЧЕНИЕ ЭЛЕКТРОКЛАПАНА 1 ПОДПИТКИ ОТОПЛЕНИЯ*)
			END_CASE
		110:(*-------------------------------------------------------------------------------------------ЗАПУСК СЕТЕВОГО КАСКАДА*)

				PUSK_KASKAD_NASOSOV_1_SETEVOY:=TRUE;


			IF WORK_KASKAD_1_SETEVOY  THEN
				KASKAD_GORELOK;(*--------------------------------------------------------------------ЗАПУСК КАСКАДА ГОРЕЛОК*)
			ELSE
				PUSK_GORELKA_1:=FALSE;
				PUSK_GORELKA_2:=FALSE;
				PUSK_GORELKA_3:=FALSE;
			END_IF
	END_CASE






ELSE(*------------------ЕСЛИ ПУСК КОТЕЛЬНАЯ НАЖАТА  И МОДУЛИ НЕ ОТВАЛИЛИСЬ ТО НАЧИНАЕМ ВЫПОЛНЯТЬ АЛГОРИТМ*)



	xDO.0:=xDO0:=FALSE;(*---------------------------------------------------------------------------------------НАСОС СЕТЕВОЙ 1*)
	xDO.1:=xDO1:=FALSE;(*---------------------------------------------------------------------------------------НАСОС СЕТЕВОЙ 2*)
(*
	xDO.2:=xDO2:=FALSE;(*----------------------------------------------------------------------------------НАСОС ВНУТРЕННИЙ 1*)
	xDO.3:=xDO3:=FALSE;(*----------------------------------------------------------------------------------НАСОС ВНУТРЕННИЙ 2*)
	xDO.4:=xDO4:=FALSE;(*-----------------------------------------------------------------------------------------НАСОС ГВС 1*)
	xDO.5:=xDO5:=FALSE;(*-----------------------------------------------------------------------------------------НАСОС ГВС 2*)
*)
	xDO.6:=xDO6:=FALSE;(*--------------------------------------------------------------------------------НАСОС ПОДПИТОЧНЫЙ 1*)
	xDO.7:=xDO7:=FALSE;(*--------------------------------------------------------------------------------НАСОС ПОДПИТОЧНЫЙ 2*)
	(*xDO.8:=xDO8:=FALSE;*)(*-----------------------------------------------------------------------НАСОС ЦИРКУЛЯЦИОННЫЙ 1*)
	(*xDO.9:=xDO9:=FALSE;*)(*-----------------------------------------------------------------------НАСОС ЦИРКУЛЯЦИОННЫЙ 2*)
	(*xDO.10:=xDO10:=FALSE;*)(*--------------------------------------------------------------------НАСОС ЦИРКУЛЯЦИОННЫЙ 3*)
	xDO.11:=xDO11:=FALSE;(*----------------------------------------------------------------------------------КОТЕЛ ТЕРМОСТАТ 1*)
	xDO.12:=xDO12:=FALSE;(*----------------------------------------------------------------------------------КОТЕЛ ТЕРМОСТАТ 2*)
	xDO.13:=xDO13:=FALSE;(*----------------------------------------------------------------------------------КОТЕЛ ТЕРМОСТАТ 3*)
	xDO.14:=xDO14:=FALSE;(*----------------------------------------------------------------------------------------------------------*)
	xDO.15:=xDO15:=FALSE;(*----------------------------------------------------------------------------------------------------------*)

	PUSK_GORELKA_1:=FALSE;
	PUSK_GORELKA_2:=FALSE;
	PUSK_GORELKA_3:=FALSE;
	PUSK_KASKAD_NASOSOV_1_SETEVOY:=FALSE;
	(*PUSK_KASKAD_NASOSOV_2_VNUTR:=FALSE;*)
	(*PUSK_KASKAD_NASOSOV_3_GVS:=FALSE;*)
	PUSK_KASKAD_NASOSOV_4_PODPITKA:=FALSE;

	STEP_MAIN:=0;
	STEP_DAVL_POKOYA:=0;
	STEP3:=0;
	STEP4:=0;
	(*
	STEP_SBROS_GVS:=0;
	STEP_SBROS_OTOPLENIYA:=0;
	*)
	STEP_PODOGREV_SECOND_GORELKA:=0;
	STEP_PODOGREV_RESERV_GORELKA:=0;
	STEP_AVARIA_PODOGREV_RESERV_GORELKA:=0;
END_IF(*----------------ЕСЛИ ПУСК КОТЕЛЬНАЯ НАЖАТА  И МОДУЛИ НЕ ОТВАЛИЛИСЬ ТО НАЧИНАЕМ ВЫПОЛНЯТЬ АЛГОРИТМ*)
END_ACTION
ACTION AVARIA_DATCHIK:
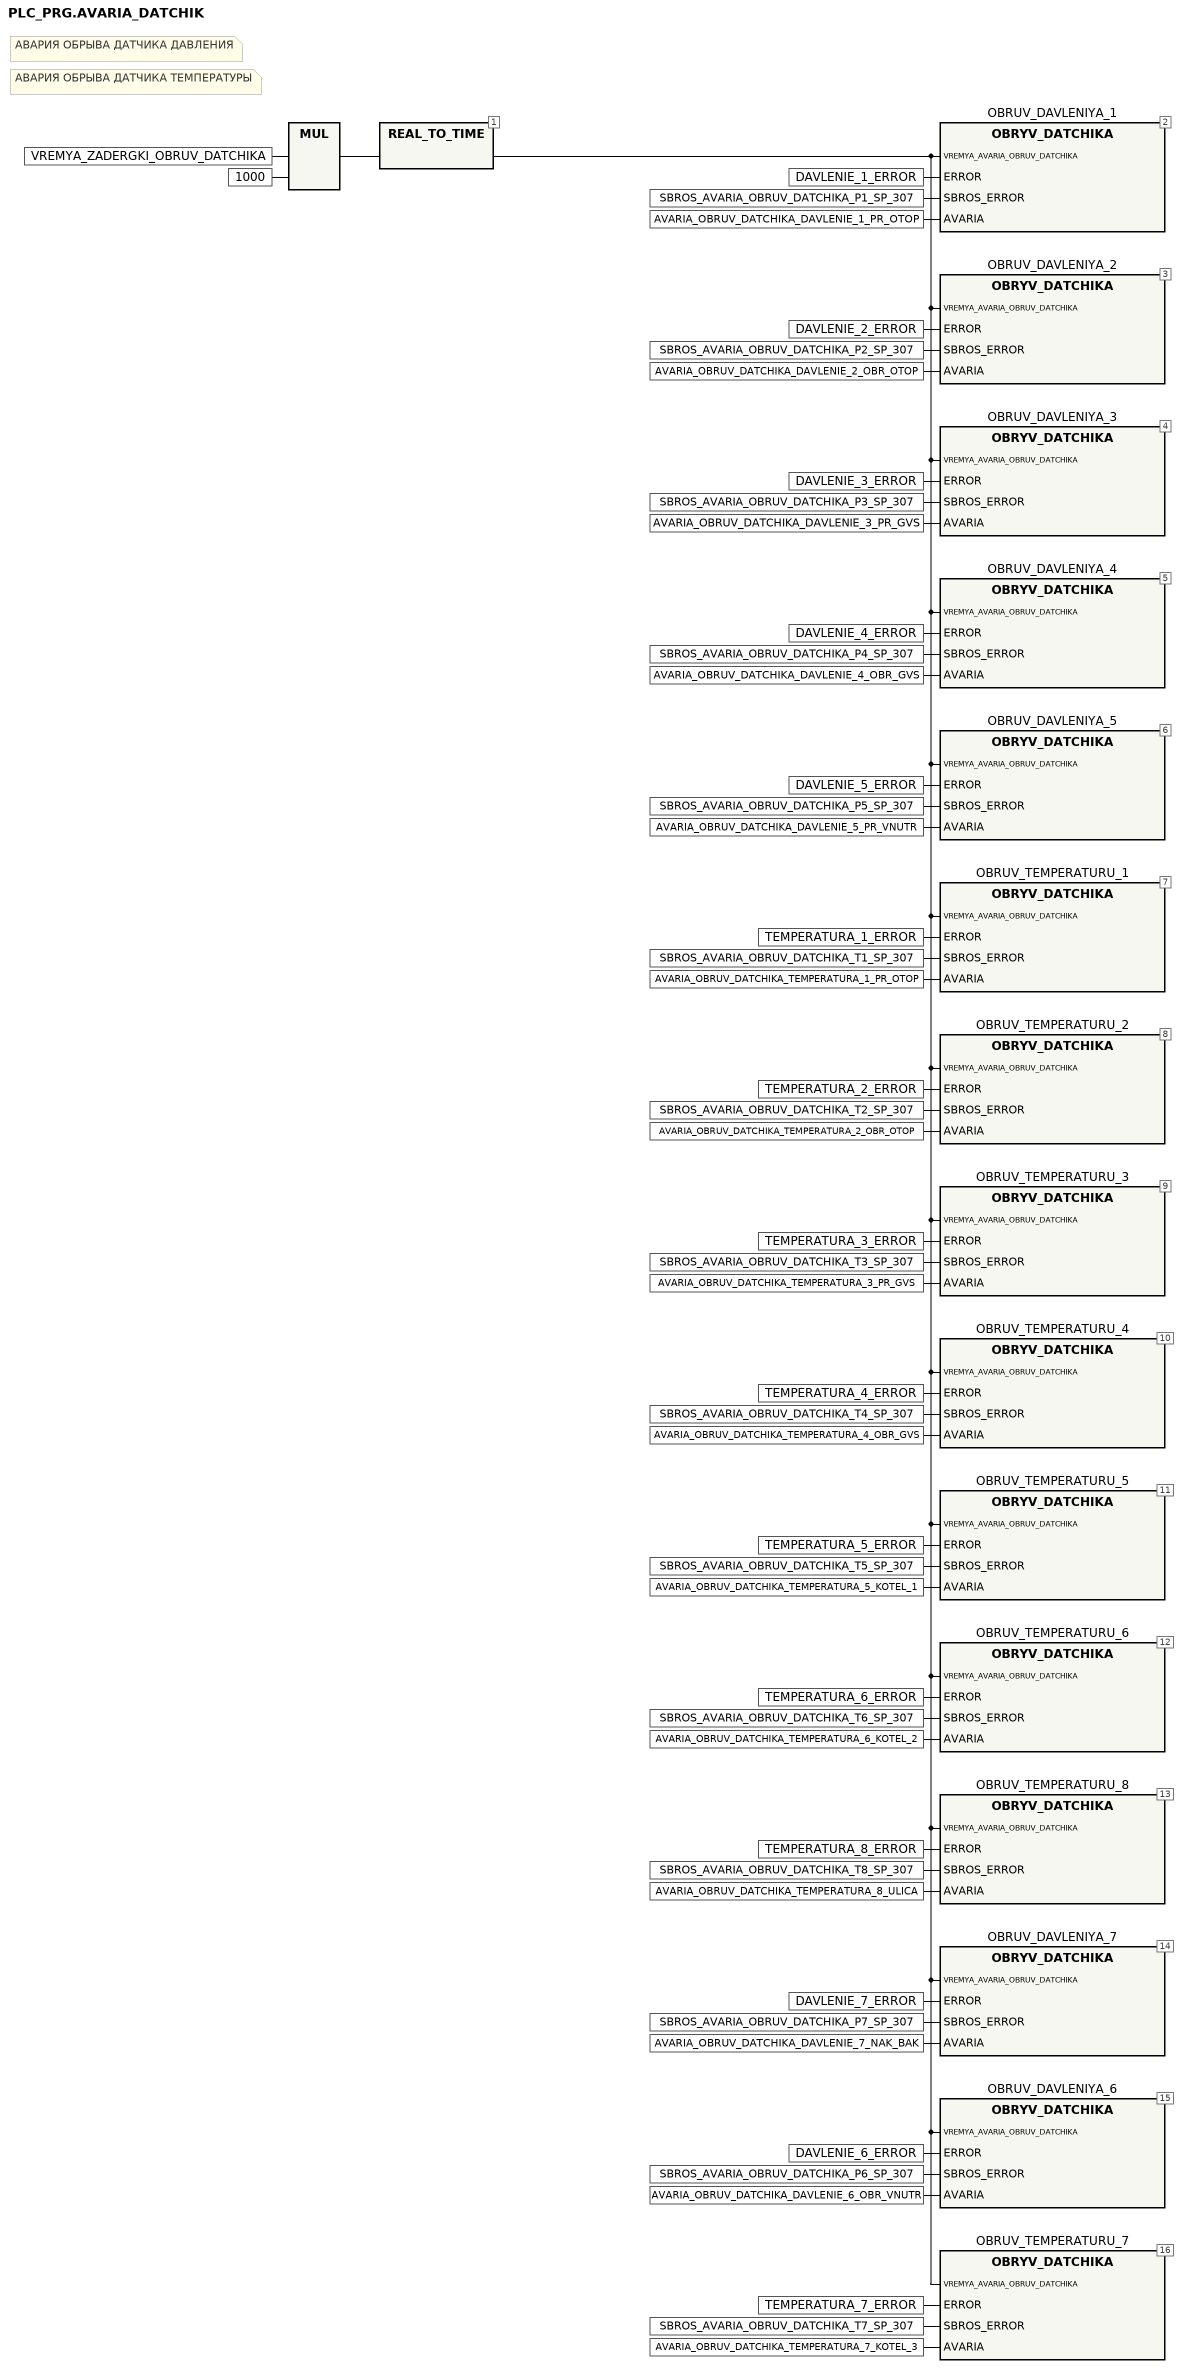
_CFC_ (* Continuous Function Chart, elements in execution order *)
#0 MUL(VREMYA_ZADERGKI_OBRUV_DATCHIKA, 1000)
#1 REAL_TO_TIME(#0)
#2 OBRUV_DAVLENIYA_1:OBRYV_DATCHIKA(VREMYA_AVARIA_OBRUV_DATCHIKA: #1, ERROR: DAVLENIE_1_ERROR, SBROS_ERROR: SBROS_AVARIA_OBRUV_DATCHIKA_P1_SP_307, AVARIA: AVARIA_OBRUV_DATCHIKA_DAVLENIE_1_PR_OTOP)
(* АВАРИЯ ОБРЫВА ДАТЧИКА ДАВЛЕНИЯ *)
#3 OBRUV_DAVLENIYA_2:OBRYV_DATCHIKA(VREMYA_AVARIA_OBRUV_DATCHIKA: #1, ERROR: DAVLENIE_2_ERROR, SBROS_ERROR: SBROS_AVARIA_OBRUV_DATCHIKA_P2_SP_307, AVARIA: AVARIA_OBRUV_DATCHIKA_DAVLENIE_2_OBR_OTOP)
#4 OBRUV_DAVLENIYA_3:OBRYV_DATCHIKA(VREMYA_AVARIA_OBRUV_DATCHIKA: #1, ERROR: DAVLENIE_3_ERROR, SBROS_ERROR: SBROS_AVARIA_OBRUV_DATCHIKA_P3_SP_307, AVARIA: AVARIA_OBRUV_DATCHIKA_DAVLENIE_3_PR_GVS)
#5 OBRUV_DAVLENIYA_4:OBRYV_DATCHIKA(VREMYA_AVARIA_OBRUV_DATCHIKA: #1, ERROR: DAVLENIE_4_ERROR, SBROS_ERROR: SBROS_AVARIA_OBRUV_DATCHIKA_P4_SP_307, AVARIA: AVARIA_OBRUV_DATCHIKA_DAVLENIE_4_OBR_GVS)
#6 OBRUV_DAVLENIYA_5:OBRYV_DATCHIKA(VREMYA_AVARIA_OBRUV_DATCHIKA: #1, ERROR: DAVLENIE_5_ERROR, SBROS_ERROR: SBROS_AVARIA_OBRUV_DATCHIKA_P5_SP_307, AVARIA: AVARIA_OBRUV_DATCHIKA_DAVLENIE_5_PR_VNUTR)
#7 OBRUV_TEMPERATURU_1:OBRYV_DATCHIKA(VREMYA_AVARIA_OBRUV_DATCHIKA: #1, ERROR: TEMPERATURA_1_ERROR, SBROS_ERROR: SBROS_AVARIA_OBRUV_DATCHIKA_T1_SP_307, AVARIA: AVARIA_OBRUV_DATCHIKA_TEMPERATURA_1_PR_OTOP)
(* АВАРИЯ ОБРЫВА ДАТЧИКА ТЕМПЕРАТУРЫ *)
#8 OBRUV_TEMPERATURU_2:OBRYV_DATCHIKA(VREMYA_AVARIA_OBRUV_DATCHIKA: #1, ERROR: TEMPERATURA_2_ERROR, SBROS_ERROR: SBROS_AVARIA_OBRUV_DATCHIKA_T2_SP_307, AVARIA: AVARIA_OBRUV_DATCHIKA_TEMPERATURA_2_OBR_OTOP)
#9 OBRUV_TEMPERATURU_3:OBRYV_DATCHIKA(VREMYA_AVARIA_OBRUV_DATCHIKA: #1, ERROR: TEMPERATURA_3_ERROR, SBROS_ERROR: SBROS_AVARIA_OBRUV_DATCHIKA_T3_SP_307, AVARIA: AVARIA_OBRUV_DATCHIKA_TEMPERATURA_3_PR_GVS)
#10 OBRUV_TEMPERATURU_4:OBRYV_DATCHIKA(VREMYA_AVARIA_OBRUV_DATCHIKA: #1, ERROR: TEMPERATURA_4_ERROR, SBROS_ERROR: SBROS_AVARIA_OBRUV_DATCHIKA_T4_SP_307, AVARIA: AVARIA_OBRUV_DATCHIKA_TEMPERATURA_4_OBR_GVS)
#11 OBRUV_TEMPERATURU_5:OBRYV_DATCHIKA(VREMYA_AVARIA_OBRUV_DATCHIKA: #1, ERROR: TEMPERATURA_5_ERROR, SBROS_ERROR: SBROS_AVARIA_OBRUV_DATCHIKA_T5_SP_307, AVARIA: AVARIA_OBRUV_DATCHIKA_TEMPERATURA_5_KOTEL_1)
#12 OBRUV_TEMPERATURU_6:OBRYV_DATCHIKA(VREMYA_AVARIA_OBRUV_DATCHIKA: #1, ERROR: TEMPERATURA_6_ERROR, SBROS_ERROR: SBROS_AVARIA_OBRUV_DATCHIKA_T6_SP_307, AVARIA: AVARIA_OBRUV_DATCHIKA_TEMPERATURA_6_KOTEL_2)
#13 OBRUV_TEMPERATURU_8:OBRYV_DATCHIKA(VREMYA_AVARIA_OBRUV_DATCHIKA: #1, ERROR: TEMPERATURA_8_ERROR, SBROS_ERROR: SBROS_AVARIA_OBRUV_DATCHIKA_T8_SP_307, AVARIA: AVARIA_OBRUV_DATCHIKA_TEMPERATURA_8_ULICA)
#14 OBRUV_DAVLENIYA_7:OBRYV_DATCHIKA(VREMYA_AVARIA_OBRUV_DATCHIKA: #1, ERROR: DAVLENIE_7_ERROR, SBROS_ERROR: SBROS_AVARIA_OBRUV_DATCHIKA_P7_SP_307, AVARIA: AVARIA_OBRUV_DATCHIKA_DAVLENIE_7_NAK_BAK)
#15 OBRUV_DAVLENIYA_6:OBRYV_DATCHIKA(VREMYA_AVARIA_OBRUV_DATCHIKA: #1, ERROR: DAVLENIE_6_ERROR, SBROS_ERROR: SBROS_AVARIA_OBRUV_DATCHIKA_P6_SP_307, AVARIA: AVARIA_OBRUV_DATCHIKA_DAVLENIE_6_OBR_VNUTR)
#16 OBRUV_TEMPERATURU_7:OBRYV_DATCHIKA(VREMYA_AVARIA_OBRUV_DATCHIKA: #1, ERROR: TEMPERATURA_7_ERROR, SBROS_ERROR: SBROS_AVARIA_OBRUV_DATCHIKA_T7_SP_307, AVARIA: AVARIA_OBRUV_DATCHIKA_TEMPERATURA_7_KOTEL_3)
_END_CFC_
(* the same logic as Structured Text *)
_t5 := REAL_TO_TIME(VREMYA_ZADERGKI_OBRUV_DATCHIKA * 1000);
OBRUV_DAVLENIYA_1(VREMYA_AVARIA_OBRUV_DATCHIKA := _t5, ERROR := DAVLENIE_1_ERROR, SBROS_ERROR := SBROS_AVARIA_OBRUV_DATCHIKA_P1_SP_307, AVARIA := AVARIA_OBRUV_DATCHIKA_DAVLENIE_1_PR_OTOP);
(* АВАРИЯ ОБРЫВА ДАТЧИКА ДАВЛЕНИЯ *)
OBRUV_DAVLENIYA_2(VREMYA_AVARIA_OBRUV_DATCHIKA := _t5, ERROR := DAVLENIE_2_ERROR, SBROS_ERROR := SBROS_AVARIA_OBRUV_DATCHIKA_P2_SP_307, AVARIA := AVARIA_OBRUV_DATCHIKA_DAVLENIE_2_OBR_OTOP);
OBRUV_DAVLENIYA_3(VREMYA_AVARIA_OBRUV_DATCHIKA := _t5, ERROR := DAVLENIE_3_ERROR, SBROS_ERROR := SBROS_AVARIA_OBRUV_DATCHIKA_P3_SP_307, AVARIA := AVARIA_OBRUV_DATCHIKA_DAVLENIE_3_PR_GVS);
OBRUV_DAVLENIYA_4(VREMYA_AVARIA_OBRUV_DATCHIKA := _t5, ERROR := DAVLENIE_4_ERROR, SBROS_ERROR := SBROS_AVARIA_OBRUV_DATCHIKA_P4_SP_307, AVARIA := AVARIA_OBRUV_DATCHIKA_DAVLENIE_4_OBR_GVS);
OBRUV_DAVLENIYA_5(VREMYA_AVARIA_OBRUV_DATCHIKA := _t5, ERROR := DAVLENIE_5_ERROR, SBROS_ERROR := SBROS_AVARIA_OBRUV_DATCHIKA_P5_SP_307, AVARIA := AVARIA_OBRUV_DATCHIKA_DAVLENIE_5_PR_VNUTR);
OBRUV_TEMPERATURU_1(VREMYA_AVARIA_OBRUV_DATCHIKA := _t5, ERROR := TEMPERATURA_1_ERROR, SBROS_ERROR := SBROS_AVARIA_OBRUV_DATCHIKA_T1_SP_307, AVARIA := AVARIA_OBRUV_DATCHIKA_TEMPERATURA_1_PR_OTOP);
(* АВАРИЯ ОБРЫВА ДАТЧИКА ТЕМПЕРАТУРЫ *)
OBRUV_TEMPERATURU_2(VREMYA_AVARIA_OBRUV_DATCHIKA := _t5, ERROR := TEMPERATURA_2_ERROR, SBROS_ERROR := SBROS_AVARIA_OBRUV_DATCHIKA_T2_SP_307, AVARIA := AVARIA_OBRUV_DATCHIKA_TEMPERATURA_2_OBR_OTOP);
OBRUV_TEMPERATURU_3(VREMYA_AVARIA_OBRUV_DATCHIKA := _t5, ERROR := TEMPERATURA_3_ERROR, SBROS_ERROR := SBROS_AVARIA_OBRUV_DATCHIKA_T3_SP_307, AVARIA := AVARIA_OBRUV_DATCHIKA_TEMPERATURA_3_PR_GVS);
OBRUV_TEMPERATURU_4(VREMYA_AVARIA_OBRUV_DATCHIKA := _t5, ERROR := TEMPERATURA_4_ERROR, SBROS_ERROR := SBROS_AVARIA_OBRUV_DATCHIKA_T4_SP_307, AVARIA := AVARIA_OBRUV_DATCHIKA_TEMPERATURA_4_OBR_GVS);
OBRUV_TEMPERATURU_5(VREMYA_AVARIA_OBRUV_DATCHIKA := _t5, ERROR := TEMPERATURA_5_ERROR, SBROS_ERROR := SBROS_AVARIA_OBRUV_DATCHIKA_T5_SP_307, AVARIA := AVARIA_OBRUV_DATCHIKA_TEMPERATURA_5_KOTEL_1);
OBRUV_TEMPERATURU_6(VREMYA_AVARIA_OBRUV_DATCHIKA := _t5, ERROR := TEMPERATURA_6_ERROR, SBROS_ERROR := SBROS_AVARIA_OBRUV_DATCHIKA_T6_SP_307, AVARIA := AVARIA_OBRUV_DATCHIKA_TEMPERATURA_6_KOTEL_2);
OBRUV_TEMPERATURU_8(VREMYA_AVARIA_OBRUV_DATCHIKA := _t5, ERROR := TEMPERATURA_8_ERROR, SBROS_ERROR := SBROS_AVARIA_OBRUV_DATCHIKA_T8_SP_307, AVARIA := AVARIA_OBRUV_DATCHIKA_TEMPERATURA_8_ULICA);
OBRUV_DAVLENIYA_7(VREMYA_AVARIA_OBRUV_DATCHIKA := _t5, ERROR := DAVLENIE_7_ERROR, SBROS_ERROR := SBROS_AVARIA_OBRUV_DATCHIKA_P7_SP_307, AVARIA := AVARIA_OBRUV_DATCHIKA_DAVLENIE_7_NAK_BAK);
OBRUV_DAVLENIYA_6(VREMYA_AVARIA_OBRUV_DATCHIKA := _t5, ERROR := DAVLENIE_6_ERROR, SBROS_ERROR := SBROS_AVARIA_OBRUV_DATCHIKA_P6_SP_307, AVARIA := AVARIA_OBRUV_DATCHIKA_DAVLENIE_6_OBR_VNUTR);
OBRUV_TEMPERATURU_7(VREMYA_AVARIA_OBRUV_DATCHIKA := _t5, ERROR := TEMPERATURA_7_ERROR, SBROS_ERROR := SBROS_AVARIA_OBRUV_DATCHIKA_T7_SP_307, AVARIA := AVARIA_OBRUV_DATCHIKA_TEMPERATURA_7_KOTEL_3);
END_ACTION
ACTION AVARIA_STATUS:
(*-------------------------------------------------------------------------------------------------------АВАРИЯ СЕТЕВОЙ НАСОС 1*)
IF AVARIA_SETEVOY_NASOS_1 THEN
	AVARIA_SETEVOY_NASOS_1_SP_307:=TRUE;
ELSE
	AVARIA_SETEVOY_NASOS_1_SP_307:=FALSE;
END_IF
(*-------------------------------------------------------------------------------------------------------АВАРИЯ СЕТЕВОЙ НАСОС 2*)
IF AVARIA_SETEVOY_NASOS_2 THEN
	AVARIA_SETEVOY_NASOS_2_SP_307:=TRUE;
ELSE
	AVARIA_SETEVOY_NASOS_2_SP_307:=FALSE;
END_IF
(*-----------------------------------------------------------------------------------------------------------АВАРИЯ ЛЕТНИЙ НАСОС*)
(*------------------------------------------------------------------------------------------------------------------------------------------------------УДАЛИТЬ
IF AVARIA_LETNIY_NASOS THEN
	AVARIA_LETNIY_NASOS_SP_307:=TRUE;
ELSE
	AVARIA_LETNIY_NASOS_SP_307:=FALSE;
END_IF
*)
(*--------------------------------------------------------------------------------------------------------------АВАРИЯ НАСОС ГВС 1*)
IF AVARIA_GVS_NASOS_1 THEN
	AVARIA_GVS_NASOS_1_SP_307:=TRUE;
ELSE
	AVARIA_GVS_NASOS_1_SP_307:=FALSE;
END_IF
(*--------------------------------------------------------------------------------------------------------------АВАРИЯ НАСОС ГВС 2*)
IF AVARIA_GVS_NASOS_2 THEN
	AVARIA_GVS_NASOS_2_SP_307:=TRUE;
ELSE
	AVARIA_GVS_NASOS_2_SP_307:=FALSE;
END_IF
(*------------------------------------------------------------------------------------------------АВАРИЯ ПОДПИТОЧНЫЙ НАСОС 1*)
IF AVARIA_PODPITOCHNYU_NASOS_1 THEN
	AVARIA_PODPITOCHNYU_NASOS_1_SP_307:=TRUE;
ELSE
	AVARIA_PODPITOCHNYU_NASOS_1_SP_307:=FALSE;
END_IF
(*------------------------------------------------------------------------------------------------АВАРИЯ ПОДПИТОЧНЫЙ НАСОС 2*)
IF AVARIA_PODPITOCHNYU_NASOS_2 THEN
	AVARIA_PODPITOCHNYU_NASOS_2_SP_307:=TRUE;
ELSE
	AVARIA_PODPITOCHNYU_NASOS_2_SP_307:=FALSE;
END_IF
(*----------------------------------------------------------------------------------------------------------------АВАРИЯ ГОРЕЛКА 1*)
IF AVARIA_GORELKA_1 THEN
	AVARIA_GORELKA_1_SP_307:=TRUE;
ELSE
	AVARIA_GORELKA_1_SP_307:=FALSE;
END_IF
(*----------------------------------------------------------------------------------------------------------------АВАРИЯ ГОРЕЛКА 2*)
IF AVARIA_GORELKA_2 THEN
	AVARIA_GORELKA_2_SP_307:=TRUE;
ELSE
	AVARIA_GORELKA_2_SP_307:=FALSE;
END_IF
(*----------------------------------------------------------------------------------------------------------------АВАРИЯ ГОРЕЛКА 3*)
IF AVARIA_GORELKA_3 THEN
	AVARIA_GORELKA_3_SP_307:=TRUE;
ELSE
	AVARIA_GORELKA_3_SP_307:=FALSE;
END_IF
(*
(*---------------------------------------------------------------------------------------- ПРЕДУПРЕЖДЕНИЕ ВКЛЮЧИТЕ ГОРЕЛКУ 1*)
IF xDO.12 AND PUSK_GORELKA_1 AND B4_GORELKA_1=FALSE THEN
	STEP_STATUS_PREDUPREGDENIE_ON_GORELKA_1:=1;
ELSE
	PREDUPREGDENIE_VKLUCHITE_GORELKU_1_SP_307:=FALSE;
	STEP_STATUS_PREDUPREGDENIE_ON_GORELKA_1:=0;
	TIMER_STATUS_PREDUPREGDENIE_ON_GORELKA_1(IN:=FALSE,PT:=T#0s);
      	TIMER_STATUS_PREDUPREGDENIE_ON_GORELKA_1;
END_IF

CASE STEP_STATUS_PREDUPREGDENIE_ON_GORELKA_1 OF
	1:
		TIMER_STATUS_PREDUPREGDENIE_ON_GORELKA_1(IN:=TRUE,
													  PT:=REAL_TO_TIME(VREMYA_ZADERGKI_AVARIA_NIZKOE_DAVLENIE*1000));
		IF  TIMER_STATUS_PREDUPREGDENIE_ON_GORELKA_1.ET=TIMER_STATUS_PREDUPREGDENIE_ON_GORELKA_1.PT THEN
			IF xDO.12 AND PUSK_GORELKA_1 AND B4_GORELKA_1=FALSE THEN

				PREDUPREGDENIE_VKLUCHITE_GORELKU_1_SP_307:=TRUE;
				STEP_STATUS_PREDUPREGDENIE_ON_GORELKA_1:=0;
				TIMER_STATUS_PREDUPREGDENIE_ON_GORELKA_1(IN:=FALSE,PT:=T#0s);
      		 		TIMER_STATUS_PREDUPREGDENIE_ON_GORELKA_1;
			ELSE
				STEP_STATUS_PREDUPREGDENIE_ON_GORELKA_1:=0;
				TIMER_STATUS_PREDUPREGDENIE_ON_GORELKA_1(IN:=FALSE,PT:=T#0s);
      		 		TIMER_STATUS_PREDUPREGDENIE_ON_GORELKA_1;
			END_IF
		END_IF
END_CASE
*)
(*
(*---------------------------------------------------------------------------------------- ПРЕДУПРЕЖДЕНИЕ ВКЛЮЧИТЕ ГОРЕЛКУ 2*)
IF xDO.13 AND PUSK_GORELKA_2 AND B4_GORELKA_2=FALSE THEN
	STEP_STATUS_PREDUPREGDENIE_ON_GORELKA_2:=1;
ELSE
	PREDUPREGDENIE_VKLUCHITE_GORELKU_2_SP_307:=FALSE;
	STEP_STATUS_PREDUPREGDENIE_ON_GORELKA_2:=0;
	TIMER_STATUS_PREDUPREGDENIE_ON_GORELKA_2(IN:=FALSE,PT:=T#0s);
      	TIMER_STATUS_PREDUPREGDENIE_ON_GORELKA_2;
END_IF


CASE STEP_STATUS_PREDUPREGDENIE_ON_GORELKA_2 OF
	1:
		TIMER_STATUS_PREDUPREGDENIE_ON_GORELKA_2(IN:=TRUE,
													  PT:=REAL_TO_TIME(VREMYA_ZADERGKI_AVARIA_NIZKOE_DAVLENIE*1000));
		IF  TIMER_STATUS_PREDUPREGDENIE_ON_GORELKA_2.ET=TIMER_STATUS_PREDUPREGDENIE_ON_GORELKA_2.PT THEN
			IF xDO.13 AND PUSK_GORELKA_2 AND B4_GORELKA_2=FALSE THEN

				PREDUPREGDENIE_VKLUCHITE_GORELKU_2_SP_307:=TRUE;
				STEP_STATUS_PREDUPREGDENIE_ON_GORELKA_2:=0;
				TIMER_STATUS_PREDUPREGDENIE_ON_GORELKA_2(IN:=FALSE,PT:=T#0s);
      		 		TIMER_STATUS_PREDUPREGDENIE_ON_GORELKA_2;
			ELSE
				STEP_STATUS_PREDUPREGDENIE_ON_GORELKA_2:=0;
				TIMER_STATUS_PREDUPREGDENIE_ON_GORELKA_2(IN:=FALSE,PT:=T#0s);
      		 		TIMER_STATUS_PREDUPREGDENIE_ON_GORELKA_2;
			END_IF
		END_IF
END_CASE
*)





(*---------------------------------------------------------------------------------------------АВАРИЯ/СБРОС РЕЛЕ КОНТРОЛЯ ФАЗ*)
IF RELE_KONTROL_PHAS=FALSE THEN
	AVARIA_PHASA_SP_307:=TRUE;
END_IF

(*------------------------------------------------------------------------------------------------------------------ОБРЫВ ДАТЧИКОВ*)
AVARIA_OBRUV_DATCHIKA_P1_SP_307:=AVARIA_OBRUV_DATCHIKA_DAVLENIE_1_PR_OTOP;
AVARIA_OBRUV_DATCHIKA_P2_SP_307:=AVARIA_OBRUV_DATCHIKA_DAVLENIE_2_OBR_OTOP;
AVARIA_OBRUV_DATCHIKA_P3_SP_307:=AVARIA_OBRUV_DATCHIKA_DAVLENIE_3_PR_GVS;
AVARIA_OBRUV_DATCHIKA_P4_SP_307:=AVARIA_OBRUV_DATCHIKA_DAVLENIE_4_OBR_GVS;

AVARIA_OBRUV_DATCHIKA_P5_SP_307:=AVARIA_OBRUV_DATCHIKA_DAVLENIE_5_PR_VNUTR;
AVARIA_OBRUV_DATCHIKA_P6_SP_307:=AVARIA_OBRUV_DATCHIKA_DAVLENIE_6_OBR_VNUTR;


AVARIA_OBRUV_DATCHIKA_P7_SP_307:=AVARIA_OBRUV_DATCHIKA_DAVLENIE_7_NAK_BAK;

AVARIA_OBRUV_DATCHIKA_T1_SP_307:=AVARIA_OBRUV_DATCHIKA_TEMPERATURA_1_PR_OTOP;
AVARIA_OBRUV_DATCHIKA_T2_SP_307:=AVARIA_OBRUV_DATCHIKA_TEMPERATURA_2_OBR_OTOP;
AVARIA_OBRUV_DATCHIKA_T3_SP_307:=AVARIA_OBRUV_DATCHIKA_TEMPERATURA_3_PR_GVS;
AVARIA_OBRUV_DATCHIKA_T4_SP_307:=AVARIA_OBRUV_DATCHIKA_TEMPERATURA_4_OBR_GVS;
AVARIA_OBRUV_DATCHIKA_T5_SP_307:=AVARIA_OBRUV_DATCHIKA_TEMPERATURA_5_KOTEL_1;
AVARIA_OBRUV_DATCHIKA_T6_SP_307:=AVARIA_OBRUV_DATCHIKA_TEMPERATURA_6_KOTEL_2;
AVARIA_OBRUV_DATCHIKA_T7_SP_307:=AVARIA_OBRUV_DATCHIKA_TEMPERATURA_7_KOTEL_3;

AVARIA_OBRUV_DATCHIKA_T8_SP_307:=AVARIA_OBRUV_DATCHIKA_TEMPERATURA_8_ULICA;


(*-------------------------------ЕСЛИ ОБРЫВ ДАТЧИКА P2 ОБРАТКИ ОТОПЛЕНИЯ УВОДИМ В АВАРИЮ ПОДПИТОЧНЫЕ НАСОСЫ*)
IF AVARIA_OBRUV_DATCHIKA_P2_SP_307  THEN
	AVARIA_PODPITOCHNYU_NASOS_1:=TRUE;
	AVARIA_PODPITOCHNYU_NASOS_2:=TRUE;
END_IF

(*--------------------------------------------------------------------ОШИБКА ГОРЕЛКИ 1 ПО ОБРЫВУ ДАТЧИКА ТЕМПЕРАТУРЫ 5*)
IF AVARIA_OBRUV_DATCHIKA_TEMPERATURA_5_KOTEL_1 THEN
	AVARIA_GORELKA_1:=TRUE;
END_IF
(*--------------------------------------------------------------------ОШИБКА ГОРЕЛКИ 2 ПО ОБРЫВУ ДАТЧИКА ТЕМПЕРАТУРЫ 6*)
IF AVARIA_OBRUV_DATCHIKA_TEMPERATURA_6_KOTEL_2 THEN
	AVARIA_GORELKA_2:=TRUE;
END_IF
(*--------------------------------------------------------------------ОШИБКА ГОРЕЛКИ 2 ПО ОБРЫВУ ДАТЧИКА ТЕМПЕРАТУРЫ 7*)
IF AVARIA_OBRUV_DATCHIKA_TEMPERATURA_7_KOTEL_3 THEN
	AVARIA_GORELKA_3:=TRUE;
END_IF
(*---------------------------------------------------------------------------------------АВАРИЯ ВЫСОКАЯ ТЕМПЕРАТУРА КОТЕЛ 1*)
IF TEMPERATURA_5_KOTEL_1_AI_SP_307>=TEMPERATURA_AVARIA_MAX_GORELKA_1 THEN
	AVARIA_VUSOKAYA_TEMPERATURA_KOTEL_1_SP_307:=TRUE;
	AVARIA_GORELKA_1:=TRUE;
END_IF

IF SBROS_AVARIA_VUSOKAYA_TEMPERATURA_KOTEL_1_SP_307=TRUE THEN
	AVARIA_VUSOKAYA_TEMPERATURA_KOTEL_1_SP_307:=FALSE;
END_IF
(*---------------------------------------------------------------------------------------АВАРИЯ ВЫСОКАЯ ТЕМПЕРАТУРА КОТЕЛ 2*)
IF TEMPERATURA_6_KOTEL_2_AI_SP_307>=TEMPERATURA_AVARIA_MAX_GORELKA_2 THEN
	AVARIA_VUSOKAYA_TEMPERATURA_KOTEL_2_SP_307:=TRUE;
	AVARIA_GORELKA_2:=TRUE;
END_IF

IF SBROS_AVARIA_VUSOKAYA_TEMPERATURA_KOTEL_2_SP_307=TRUE THEN
	AVARIA_VUSOKAYA_TEMPERATURA_KOTEL_2_SP_307:=FALSE;
END_IF
(*---------------------------------------------------------------------------------------АВАРИЯ ВЫСОКАЯ ТЕМПЕРАТУРА КОТЕЛ 3*)
IF TEMPERATURA_7_KOTEL_3_AI_SP_307>=TEMPERATURA_AVARIA_MAX_GORELKA_3 THEN
	AVARIA_VUSOKAYA_TEMPERATURA_KOTEL_3_SP_307:=TRUE;
	AVARIA_GORELKA_3:=TRUE;
END_IF

IF SBROS_AVARIA_VUSOKAYA_TEMPERATURA_KOTEL_3_SP_307=TRUE THEN
	AVARIA_VUSOKAYA_TEMPERATURA_KOTEL_3_SP_307:=FALSE;
END_IF
(*----------------------------------------------------------------------------АВАРИЯ ВЫСОКОЕ ДАВЛЕНИЕ ПРЯМОЙ ОТОПЛЕНИЯ*)
IF DAVLENIE_1_PR_OTOPLENIYA_AI_SP_307>=AVAR_DAVL_PR_OTOP_MAX AND WORK_KASKAD_1_SETEVOY THEN
	AVARIA_VUSOKOE_DAVLENIE_OTOPLENIYA_SP_307:=TRUE;
END_IF

IF SBROS_AVARIA_VUSOKOE_DAVLENIE_OTOPLENIYA_SP_307=TRUE THEN
	AVARIA_VUSOKOE_DAVLENIE_OTOPLENIYA_SP_307:=FALSE;
END_IF
(*------------------------------------------------------------------------------АВАРИЯ НИЗКОЕ ДАВЛЕНИЕ ПРЯМОЙ ОТОПЛЕНИЯ*)
IF DAVLENIE_1_PR_OTOPLENIYA_AI_SP_307<=AVAR_DAVL_PR_OTOP_MIN AND WORK_KASKAD_1_SETEVOY THEN
	STEP_AVARIA_NIZKOE_DAVLENIE_SETEVOY:=1;
ELSE
	STEP_AVARIA_NIZKOE_DAVLENIE_SETEVOY:=0;
	TIMER_AVARIA_NIZKOE_DAVLENIE_SETEVOY(IN:=FALSE,PT:=T#0s);
      	TIMER_AVARIA_NIZKOE_DAVLENIE_SETEVOY;
END_IF

CASE STEP_AVARIA_NIZKOE_DAVLENIE_SETEVOY OF
	1:
		TIMER_AVARIA_NIZKOE_DAVLENIE_SETEVOY(IN:=TRUE,
													  PT:=REAL_TO_TIME(VREMYA_ZADERGKI_AVARIA_NIZKOE_DAVLENIE*1000));
		IF  TIMER_AVARIA_NIZKOE_DAVLENIE_SETEVOY.ET=TIMER_AVARIA_NIZKOE_DAVLENIE_SETEVOY.PT THEN
			IF DAVLENIE_1_PR_OTOPLENIYA_AI_SP_307<=AVAR_DAVL_PR_OTOP_MIN AND
																									WORK_KASKAD_1_SETEVOY THEN
				AVARIA_NIZKOE_DAVLENIE_OTOPLENIYA_SP_307:=TRUE;
				STEP_AVARIA_NIZKOE_DAVLENIE_SETEVOY:=0;
				TIMER_AVARIA_NIZKOE_DAVLENIE_SETEVOY(IN:=FALSE,PT:=T#0s);
      		 		TIMER_AVARIA_NIZKOE_DAVLENIE_SETEVOY;
			ELSE
				STEP_AVARIA_NIZKOE_DAVLENIE_SETEVOY:=0;
				TIMER_AVARIA_NIZKOE_DAVLENIE_SETEVOY(IN:=FALSE,PT:=T#0s);
      		 		TIMER_AVARIA_NIZKOE_DAVLENIE_SETEVOY;
			END_IF
		END_IF
END_CASE

IF SBROS_AVARIA_NIZKOE_DAVLENIE_OTOPLENIYA_SP_307=TRUE THEN
	AVARIA_NIZKOE_DAVLENIE_OTOPLENIYA_SP_307:=FALSE;
END_IF
(*------------------------------------------------------------------------------------------------АВАРИЯ ВЫСОКОЕ ДАВЛЕНИЕ ГВС*)
IF DAVLENIE_3_PR_GVS_AI_SP_307>=AVAR_DAVL_PR_GVS_MAX AND WORK_KASKAD_3_GVS THEN
	AVARIA_VUSOKOE_DAVLENIE_GVS_SP_307:=TRUE;
END_IF

IF SBROS_AVARIA_VUSOKOE_DAVLENIE_GVS_SP_307=TRUE THEN
	AVARIA_VUSOKOE_DAVLENIE_GVS_SP_307:=FALSE;
END_IF
(*--------------------------------------------------------------------------------------------------АВАРИЯ НИЗКОЕ ДАВЛЕНИЕ ГВС*)
IF DAVLENIE_3_PR_GVS_AI_SP_307<=AVAR_DAVL_PR_GVS_MIN AND WORK_KASKAD_3_GVS THEN
	STEP_AVARIA_NIZKOE_DAVLENIE_GVS:=1;
ELSE
	STEP_AVARIA_NIZKOE_DAVLENIE_GVS:=0;
	TIMER_AVARIA_NIZKOE_DAVLENIE_GVS(IN:=FALSE,PT:=T#0s);
      	TIMER_AVARIA_NIZKOE_DAVLENIE_GVS;
END_IF

CASE STEP_AVARIA_NIZKOE_DAVLENIE_GVS OF
	1:
		TIMER_AVARIA_NIZKOE_DAVLENIE_GVS(IN:=TRUE,
													  PT:=REAL_TO_TIME(VREMYA_ZADERGKI_AVARIA_NIZKOE_DAVLENIE*1000));
		IF  TIMER_AVARIA_NIZKOE_DAVLENIE_GVS.ET=TIMER_AVARIA_NIZKOE_DAVLENIE_GVS.PT THEN
			IF DAVLENIE_3_PR_GVS_AI_SP_307<=AVAR_DAVL_PR_GVS_MIN AND WORK_KASKAD_3_GVS THEN
				AVARIA_NIZKOE_DAVLENIE_GVS_SP_307:=TRUE;
				STEP_AVARIA_NIZKOE_DAVLENIE_GVS:=0;
				TIMER_AVARIA_NIZKOE_DAVLENIE_GVS(IN:=FALSE,PT:=T#0s);
      		 		TIMER_AVARIA_NIZKOE_DAVLENIE_GVS;
			ELSE
				STEP_AVARIA_NIZKOE_DAVLENIE_GVS:=0;
				TIMER_AVARIA_NIZKOE_DAVLENIE_GVS(IN:=FALSE,PT:=T#0s);
      		 		TIMER_AVARIA_NIZKOE_DAVLENIE_GVS;
			END_IF
		END_IF
END_CASE

IF SBROS_AVARIA_NIZKOE_DAVLENIE_GVS_SP_307=TRUE THEN
	AVARIA_NIZKOE_DAVLENIE_GVS_SP_307:=FALSE;
END_IF

IF STATUS_BAK_PROCENT_ZAPOLNENIA<BAK_MIN_PROCENT_AVARIA THEN
	AVARIA_NAKOPITELNUY_BAK_SP_307:=TRUE;
END_IF


IF ERROR_MODUL_SP_307 THEN
	AVARIA_MODUL_SP_307:=TRUE;
END_IF

IF  AVARIA_FIRE THEN
	AVARIA_FIRE_SP_307:=TRUE;
END_IF

IF  AVARIA_GAZ THEN
	AVARIA_GAZ_SP_307:=TRUE;
END_IF
END_ACTION
ACTION CIRCULAYCIONNYE_NASOSU:
CIRKULYACIONIY_NASOS_1;
CIRKULYACIONIY_NASOS_2;
CIRKULYACIONIY_NASOS_3;



(*(*--------------------------------------------------------------------------------------------------------ЦИРКУЛЯЦИОННЫЙ НАСОС 1*)
IF PUSK_GORELKA_1 THEN
	IF OSNOVNAYA_GORELKA=1 OR AVARIA_GORELKA_2 THEN
		xDO8:=TRUE;
	ELSE
		IF TEMPERATURA_2_OBR_OTOPLENIYA_AI_SP_307<TEMPERATURA_OFF_CIRCULACIONNOGO_NASOSA THEN
			xDO8:=TRUE;
		ELSE
			xDO8:=FALSE;
		END_IF
	END_IF
	STEP_CIRCULAYCIONNUY_NASOS_1:=1;
END_IF

IF PUSK_GORELKA_1=FALSE AND STEP_CIRCULAYCIONNUY_NASOS_1=1 THEN
	CASE STEP_CIRCULAYCIONNUY_NASOS_1 OF
		1:
			TIMER_CIRCUL_NASOS_1(IN:=TRUE,PT:=REAL_TO_TIME(VREMYA_RABOTU_CIRCULYACIONNOGO_NASOSA*1000));
				IF  TIMER_CIRCUL_NASOS_1.ET=TIMER_CIRCUL_NASOS_1.PT THEN
					STEP_CIRCULAYCIONNUY_NASOS_1:=0;
					TIMER_CIRCUL_NASOS_1(IN:=FALSE,PT:=T#0s);
      		 			TIMER_CIRCUL_NASOS_1;
					xDO8:=FALSE;
				END_IF
	END_CASE
ELSE
	TIMER_CIRCUL_NASOS_1(IN:=FALSE,PT:=T#0s);
      	TIMER_CIRCUL_NASOS_1;
END_IF
(*--------------------------------------------------------------------------------------------------------ЦИРКУЛЯЦИОННЫЙ НАСОС 2*)
IF PUSK_GORELKA_2 THEN
	IF OSNOVNAYA_GORELKA=2 OR AVARIA_GORELKA_1 THEN
		xDO9:=TRUE;
	ELSE
		IF TEMPERATURA_2_OBR_OTOPLENIYA_AI_SP_307<TEMPERATURA_OFF_CIRCULACIONNOGO_NASOSA THEN
			xDO9:=TRUE;
		ELSE
			xDO9:=FALSE;
		END_IF
	END_IF
	STEP_CIRCULAYCIONNUY_NASOS_2:=1;
END_IF

IF PUSK_GORELKA_2=FALSE AND STEP_CIRCULAYCIONNUY_NASOS_2=1 THEN
	CASE STEP_CIRCULAYCIONNUY_NASOS_2 OF
		1:
			TIMER_CIRCUL_NASOS_2(IN:=TRUE,PT:=REAL_TO_TIME(VREMYA_RABOTU_CIRCULYACIONNOGO_NASOSA*1000));
				IF  TIMER_CIRCUL_NASOS_2.ET=TIMER_CIRCUL_NASOS_2.PT THEN
					STEP_CIRCULAYCIONNUY_NASOS_2:=0;
					TIMER_CIRCUL_NASOS_2(IN:=FALSE,PT:=T#0s);
      		 			TIMER_CIRCUL_NASOS_2;
					xDO9:=FALSE;
				END_IF
	END_CASE
ELSE
	TIMER_CIRCUL_NASOS_2(IN:=FALSE,PT:=T#0s);
      	TIMER_CIRCUL_NASOS_2;
END_IF
(*--------------------------------------------------------------------------------------------------------ЦИРКУЛЯЦИОННЫЙ НАСОС 3*)
IF PUSK_GORELKA_3 THEN
	IF OSNOVNAYA_GORELKA=3 OR AVARIA_GORELKA_3 THEN
		xDO10:=TRUE;
	ELSE
		IF TEMPERATURA_2_OBR_OTOPLENIYA_AI_SP_307<TEMPERATURA_OFF_CIRCULACIONNOGO_NASOSA THEN
			xDO10:=TRUE;
		ELSE
			xDO10:=FALSE;
		END_IF
	END_IF
	STEP_CIRCULAYCIONNUY_NASOS_3:=1;
END_IF

IF PUSK_GORELKA_3=FALSE AND STEP_CIRCULAYCIONNUY_NASOS_3=1 THEN
	CASE STEP_CIRCULAYCIONNUY_NASOS_3 OF
		1:
			TIMER_CIRCUL_NASOS_3(IN:=TRUE,PT:=REAL_TO_TIME(VREMYA_RABOTU_CIRCULYACIONNOGO_NASOSA*1000));
				IF  TIMER_CIRCUL_NASOS_3.ET=TIMER_CIRCUL_NASOS_3.PT THEN
					STEP_CIRCULAYCIONNUY_NASOS_3:=0;
					TIMER_CIRCUL_NASOS_3(IN:=FALSE,PT:=T#0s);
      		 			TIMER_CIRCUL_NASOS_3;
					xDO10:=FALSE;
				END_IF
	END_CASE
ELSE
	TIMER_CIRCUL_NASOS_3(IN:=FALSE,PT:=T#0s);
      	TIMER_CIRCUL_NASOS_3;
END_IF
*)
END_ACTION
ACTION CIRKULYACIONIY_NASOS_1:
IF PUSK_GORELKA_1=TRUE  THEN
(*---------------------------------------------------------------------------------------------------ЕСЛИ ОСНОВНАЯ ГОРЕЛКА 1*)
	IF  OSNOVNAYA_GORELKA=1  THEN
		xDO8:=TRUE;
		STEP_CIRCULAYCIONNUY_NASOS_1:=1;
	END_IF

